	TblTemplate.InsertHParam(Table:= Table);          	
	Error													:= TblTemplate.Error;
	ErrorId													:= TblTemplate.ErrorId;
	ErrorText												:= TblTemplate.ErrorText;
	FilledRows												:= TblTemplate.FilledRows;
	
	SetHParam												:= NOT Error;
(*************************************************************************************)
END_METHOD

METHOD setPathDynamics : BOOL //Return value = TRUE if executed succesful
VAR_INPUT
	Acc,Dec,Jerk											:	LREAL;
END_VAR
	(* NCI SetPathDynamics schreiben						*)
	(*********************************************************)

(* Zielpos. in Tabelle schreiben ************************************************************)
	BlockCount 												:= BlockCount + 1;
	TblTemplate.PathDynamics.nDisplayIndex := LastBlockNo := SEL(BlockNo = 0, BlockNo, TableNumber * OffsetFactorTblNumber + BlockCount);

	TblTemplate.PathDynamics.fDec							:= Dec;
	TblTemplate.PathDynamics.fJerk							:= Jerk;
	TblTemplate.PathDynamics.fAcc							:= Acc;
                                                        	
	TblTemplate.InsertPathDynamics(Table:= Table);    	
	Error													:= TblTemplate.Error;
	ErrorId													:= TblTemplate.ErrorId;
	ErrorText												:= TblTemplate.ErrorText;
	FilledRows												:= TblTemplate.FilledRows;

	SetPathDynamics											:= NOT Error;
(***************************************************************************)
END_METHOD

METHOD setSParam : bool //Return value = TRUE if executed succesful
VAR_INPUT
	SParam													: UINT;
END_VAR
(* 														*)
(********************************************************)

(*************************************************************************************)
	BlockCount 												:= BlockCount + 1;
	TblTemplate.SParam.nDisplayIndex := LastBlockNo 		:= SEL(BlockNo = 0, BlockNo,  TableNumber * OffsetFactorTblNumber + BlockCount);
	TblTemplate.SParam.nSParam								:= SParam;
                                                        	
	TblTemplate.InsertSParam(Table:= Table);          	
	Error													:= TblTemplate.Error;
	ErrorId													:= TblTemplate.ErrorId;
	ErrorText												:= TblTemplate.ErrorText;
	FilledRows												:= TblTemplate.FilledRows;
	
	SetSParam												:= NOT Error;
(*************************************************************************************)
END_METHOD

METHOD setTangFollowingDesc : booL //Return value = TRUE if executed succesful
VAR_INPUT
    TangOn													: BOOL;
    TangAxis												: E_NciAxesInGroup;  
    PathAxis1												: E_NciAxesInGroup; 
    PathAxis2												: E_NciAxesInGroup; 
    Offset													: LREAL; 
    CriticalAngle1											: LREAL;
    TfBehavior												: E_TangentialFollowingBehavior; 
END_VAR
	(* NCI SetTangFollowingDesc schreiben						*)
	(*********************************************************)

(* Zielpos. in Tabelle schreiben ************************************************************)
	BlockCount 												:= BlockCount + 1;
	LastBlockNo 											:= SEL(BlockNo = 0, BlockNo, TableNumber * OffsetFactorTblNumber + BlockCount);

    TblTemplate.TangentialFollowingDesc.bTangOn				:= TangOn;
    TblTemplate.TangentialFollowingDesc.nTangAxis			:= TangAxis;
    TblTemplate.TangentialFollowingDesc.nPathAxis1			:= PathAxis1;
    TblTemplate.TangentialFollowingDesc.nPathAxis2			:= PathAxis2;
    TblTemplate.TangentialFollowingDesc.fOffset				:= Offset;
    TblTemplate.TangentialFollowingDesc.fCriticalAngle1		:= CriticalAngle1;
    TblTemplate.TangentialFollowingDesc.nTfBehavior			:= TfBehavior;
                       	
	TblTemplate.InsertTangFollowingDesc(Table:= Table);    	
	Error													:= TblTemplate.Error;
	ErrorId													:= TblTemplate.ErrorId;
	ErrorText												:= TblTemplate.ErrorText;
	FilledRows												:= TblTemplate.FilledRows;

	SetTangFollowingDesc									:= NOT Error;
(***************************************************************************)
END_METHOD

METHOD setTParam : bool //Return value = TRUE if executed succesful
VAR_INPUT
	TParam													: UINT;
END_VAR
(* 														*)
(********************************************************)

(*************************************************************************************)
	BlockCount 												:= BlockCount + 1;
	TblTemplate.TParam.nDisplayIndex := LastBlockNo 		:= SEL(BlockNo = 0, BlockNo,  TableNumber * OffsetFactorTblNumber + BlockCount);
	TblTemplate.TParam.nTParam								:= TParam;
                                                        	
	TblTemplate.InsertTParam(Table:= Table);          	
	Error													:= TblTemplate.Error;
	ErrorId													:= TblTemplate.ErrorId;
	ErrorText												:= TblTemplate.ErrorText;
	FilledRows												:= TblTemplate.FilledRows;
	
	SetTParam												:= NOT Error;
(**************************************************************************)
END_METHOD

METHOD setVertexSmoothing : BOOL //Return value = TRUE if executed succesful
VAR_INPUT
	Radius													: LREAL := 0.0;
	VertSmType												: UDINT := 5;
	VertSmSubType											: UDINT := 3;
END_VAR
(* writing NCI Vertex smoothing 								*)
(****************************************************************)

(* writing into table	*****************************************)
	BlockCount 												:= BlockCount + 1;
	TblTemplate.VertexSmoothing.nDisplayIndex := LastBlockNo := SEL(BlockNo = 0, BlockNo, TableNumber * OffsetFactorTblNumber + BlockCount);
	TblTemplate.VertexSmoothing.nType						:= VertSmType;
	TblTemplate.VertexSmoothing.nSubtype					:= VertSmSubtype; (* 	1: constant radius tolerance
																					2: distance between Abstand intersectoin point and peal point
																					3: adaptiv raidus tolerance
																					*)
	TblTemplate.VertexSmoothing.fRadius						:= Radius; (* mm *)

	TblTemplate.InsertVertexSmoothing(Table:= Table);
	Error													:= TblTemplate.Error;
	ErrorId													:= TblTemplate.ErrorId;
	ErrorText												:= TblTemplate.ErrorText;
	FilledRows												:= TblTemplate.FilledRows;
	SetVertexSmoothing										:= not Error;
(*************************************************************************************)
END_METHOD

END_FUNCTION_BLOCK

// POUs/Motion/TF5100-NCI/02_Options/PlcItp/NciCreateItpTableEntryTemplate
FUNCTION_BLOCK NciCreateItpTableEntryTemplate
VAR_INPUT
	EndOfTables												: ST_NciEndOfTables;
	GeoCirclePlane											: ST_NciGeoCirclePlane;
	GeoCircleCIP											: ST_NciGeoCircleCIP;
	GeoLine													: ST_NciGeoLine;
	GeoBezier3												: ST_NciGeoBezier3;
	GeoBezier5												: ST_NciGeoBezier5;	
	GeoStart												: ST_NciGeoStart;
	TangentialFollowingDesc									: ST_NciTangentialFollowingDesc;
	MFuncHsk												: ST_NciMFuncHsk;
	MFuncFast												: ST_NciMFuncFast;
	MFuncResetAllFast										: ST_NciMFuncResetAllFast;
	HParam													: ST_NciHParam;
	SParam													: ST_NciSParam;
	TParam													: ST_NciTParam;
	DynOverride												: ST_NciDynOvr;
	VertexSmoothing											: ST_NciVertexSmoothing;
	PathDynamics											: ST_NciPathDynamics;
	BaseFrame												: ST_NciBaseFrame;
	SetCoordinateSystem										: ST_NciSetCoordinateSystem;
	AxisDynamics											: ST_NciAxisDynamics;
	DwellTime												: ST_NciDwellTime;
END_VAR
VAR_OUTPUT
	FilledRows												: INT;
	Error													: BOOL;
{attribute 'displaymode':='hex'}
	ErrorId													: UDINT;
	ErrorText												: STRING(20);
END_VAR                 									
VAR                     									
	TblPrep													: FB_NciFeedTablePreparation;
END_VAR

(* NCI Table entry template				 	V2.0	*)
(****************************************************)

(******************************************************************************)
;
(******************************************************************************)

METHOD insertAxisDynamics : bool //Return value = TRUE if executed succesful
VAR_IN_OUT
	Table													: ST_NciFeedGroupTable;
END_VAR
	TblPrep(
		nEntryType			:= AxisDynamics.nEntryType,
		pEntry				:= ADR(AxisDynamics),
		stFeedGroupTable	:= Table,
		nFilledRows			=> FilledRows,
		bError				=> ,
		nErrorId			=> );

	IF TblPrep.bError 
	THEN
		Error												:= TRUE;
		ErrorText											:= CONCAT('AxisDynamics - JobNo. :',UDINT_TO_STRING(AxisDynamics.nDisplayIndex));
		ErrorId												:= TblPrep.nErrorId;
	ELSE
		insertAxisDynamics									:= TRUE;
	END_IF
END_METHOD

METHOD insertBaseFrame : bool //Return value = TRUE if executed succesful
VAR_IN_OUT
	Table													: ST_NciFeedGroupTable;
END_VAR
	TblPrep(
		nEntryType		:= BaseFrame.nEntryType,
		pEntry			:= ADR(BaseFrame),
		stFeedGroupTable:= Table,
		nFilledRows		=> FilledRows,
		bError			=> ,
		nErrorId		=> );

	IF TblPrep.bError 
	THEN
		Error												:= TRUE;
		ErrorText											:= CONCAT('BaseFrame - JobNo. :',UDINT_TO_STRING(BaseFrame.nDisplayIndex));
		ErrorId												:= TblPrep.nErrorId;
	ELSE
		insertBaseFrame										:= TRUE;
	END_IF
END_METHOD

METHOD insertDwellTime : booL //Return value = TRUE if executed succesful
VAR_IN_OUT
	Table													: ST_NciFeedGroupTable;
END_VAR
	TblPrep(
		nEntryType		:= DwellTime.nEntryType,
		pEntry			:= ADR(DwellTime),
		stFeedGroupTable:= Table,
		nFilledRows		=> FilledRows,
		bError			=> ,
		nErrorId		=> );

	IF TblPrep.bError 
	THEN
		Error												:= TRUE;
		ErrorText											:= CONCAT('DwellTime - JobNo. :',UDINT_TO_STRING(DwellTime.nDisplayIndex));
		ErrorId												:= TblPrep.nErrorId;
	ELSE
		insertDwellTime										:= TRUE;
	END_IF
END_METHOD

METHOD insertDynOverride : booL //Return value = TRUE if executed succesful
VAR_IN_OUT
	Table													: ST_NciFeedGroupTable;
END_VAR
	TblPrep(
		nEntryType			:= DynOverride.nEntryType,
		pEntry				:= ADR(DynOverride),
		stFeedGroupTable	:= Table,
		nFilledRows			=> FilledRows,
		bError				=> ,
		nErrorId			=> );

	IF TblPrep.bError THEN
		Error												:= TRUE;
		ErrorText											:= CONCAT('DynOverride - JobNo. :',UDINT_TO_STRING(DynOverride.nDisplayIndex));
		ErrorId												:= TblPrep.nErrorId;
	ELSE
		insertDynOverride									:= TRUE;
	END_IF
END_METHOD

METHOD insertEndOfTable : bool //Return value = TRUE if executed succesful
VAR_IN_OUT
	Table													: ST_NciFeedGroupTable;
END_VAR
	TblPrep(
		nEntryType			:= EndOfTables.nEntryType,
		pEntry				:= ADR(EndOfTables),
		stFeedGroupTable	:= Table,
		nFilledRows			=> FilledRows,
		bError				=> ,
		nErrorId			=> );

	IF TblPrep.bError THEN
		Error												:= TRUE;
		ErrorText											:= CONCAT('EndOfTables - FilledRows :',INT_TO_STRING(FilledRows));
		ErrorId												:= TblPrep.nErrorId;
	ELSE
		insertEndOfTable									:= TRUE;
	END_IF
END_METHOD

METHOD insertGeoBezier3 : booL //Return value = TRUE if executed succesful
VAR_IN_OUT
	Table													: ST_NciFeedGroupTable;
END_VAR
	TblPrep(
		nEntryType			:= GeoBezier3.nEntryType,
		pEntry				:= ADR(GeoBezier3),
		stFeedGroupTable	:= Table,
		nFilledRows			=> FilledRows,
		bError				=> ,
		nErrorId			=> );

	IF TblPrep.bError THEN
		Error												:= TRUE;
		ErrorText											:= CONCAT('GeoBezier3 - JobNo. :',UDINT_TO_STRING(GeoBezier3.nDisplayIndex));
		ErrorId												:= TblPrep.nErrorId;
	ELSE
		insertGeoBezier3									:= TRUE;
	END_IF
END_METHOD

METHOD insertGeoBezier5 : booL //Return value = TRUE if executed succesful
VAR_IN_OUT
	Table													: ST_NciFeedGroupTable;
END_VAR
	TblPrep(
		nEntryType			:= GeoBezier5.nEntryType,
		pEntry				:= ADR(GeoBezier5),
		stFeedGroupTable	:= Table,
		nFilledRows			=> FilledRows,
		bError				=> ,
		nErrorId			=> );

	IF TblPrep.bError THEN
		Error												:= TRUE;
		ErrorText											:= CONCAT('GeoBezier5 - JobNo. :',UDINT_TO_STRING(GeoBezier5.nDisplayIndex));
		ErrorId												:= TblPrep.nErrorId;
	ELSE
		insertGeoBezier5									:= TRUE;
	END_IF
END_METHOD

METHOD insertGeoCircleCIP : booL //Return value = TRUE if executed succesful
VAR_IN_OUT
	Table													: ST_NciFeedGroupTable;
END_VAR
	TblPrep(
		nEntryType			:= GeoCircleCIP.nEntryType,
		pEntry				:= ADR(GeoCircleCIP),
		stFeedGroupTable	:= Table,
		nFilledRows			=> FilledRows,
		bError				=> ,
		nErrorId			=> );

	IF TblPrep.bError 
	THEN
		Error												:= TRUE;
		ErrorText											:= CONCAT('GeoCircleCIP - JobNo. :',UDINT_TO_STRING(GeoCirclePlane.nDisplayIndex));
		ErrorId												:= TblPrep.nErrorId;
	ELSE
		insertGeoCircleCIP									:= TRUE;
	END_IF
END_METHOD

METHOD insertGeoCirclePlane : BOOL //Return value = TRUE if executed succesful
VAR_IN_OUT
	Table													: ST_NciFeedGroupTable;
END_VAR
	TblPrep(
		nEntryType			:= GeoCirclePlane.nEntryType,
		pEntry				:= ADR(GeoCirclePlane),
		stFeedGroupTable	:= Table,
		nFilledRows			=> FilledRows,
		bError				=> ,
		nErrorId			=> );

	IF TblPrep.bError 
	THEN
		Error												:= TRUE;
		ErrorText											:= CONCAT('GeoCirclePlane - JobNo. :',UDINT_TO_STRING(GeoCirclePlane.nDisplayIndex));
		ErrorId												:= TblPrep.nErrorId;
	ELSE
		insertGeoCirclePlane								:= TRUE;
	END_IF
END_METHOD

METHOD insertGeoLine : boOL //Return value = TRUE if executed succesful
VAR_IN_OUT
	Table													: ST_NciFeedGroupTable;
END_VAR
	TblPrep(
		nEntryType			:= GeoLine.nEntryType,
		pEntry				:= ADR(GeoLine),
		stFeedGroupTable	:= Table,
		nFilledRows			=> FilledRows,
		bError				=> ,
		nErrorId			=> );

	IF TblPrep.bError 
	THEN
		Error												:= TRUE;
		ErrorText											:= CONCAT('GeoLine - JobNo. :',UDINT_TO_STRING(GeoLine.nDisplayIndex));
		ErrorId												:= TblPrep.nErrorId;
	ELSE
		insertGeoLine										:= TRUE;
	END_IF
END_METHOD

METHOD insertGeoStart : booL //Return value = TRUE if executed succesful
VAR_IN_OUT
	Table													: ST_NciFeedGroupTable;
END_VAR
	TblPrep(
		nEntryType			:= GeoStart.nEntryType,
		pEntry				:= ADR(GeoStart),
		stFeedGroupTable	:= Table,
		nFilledRows			=> FilledRows,
		bError				=> ,
		nErrorId			=> );

	IF TblPrep.bError 
	THEN
		Error												:= TRUE;
		ErrorText											:= CONCAT('GeoStart - FilledRows. :',INT_TO_STRING(FilledRows));
		ErrorId												:= TblPrep.nErrorId;
	ELSE
		insertGeoStart										:= TRUE;
	END_IF
END_METHOD

METHOD insertHParam : booL //Return value = TRUE if executed succesful
VAR_IN_OUT
	Table													: ST_NciFeedGroupTable;
END_VAR
	TblPrep(
		nEntryType			:= HParam.nEntryType,
		pEntry				:= ADR(HParam),
		stFeedGroupTable	:= Table,
		nFilledRows			=> FilledRows,
		bError				=> ,
		nErrorId			=> );

	IF TblPrep.bError 
	THEN
		Error												:= TRUE;
		ErrorText											:= CONCAT('HParam - JobNo. :',UDINT_TO_STRING(HParam.nDisplayIndex));
		ErrorId												:= TblPrep.nErrorId;
	ELSE
		insertHParam										:= TRUE;
	END_IF
END_METHOD

METHOD insertMFuncFast : booL //Return value = TRUE if executed succesful
VAR_IN_OUT
	Table													: ST_NciFeedGroupTable;
END_VAR
	TblPrep(
		nEntryType			:= MFuncFast.nEntryType,
		pEntry				:= ADR(MFuncFast),
		stFeedGroupTable	:= Table,
		nFilledRows			=> FilledRows,
		bError				=> ,
		nErrorId			=> );

	IF TblPrep.bError 
	THEN
		Error												:= TRUE;
		ErrorText											:= CONCAT('MFuncFastList - JobNo. :',UDINT_TO_STRING(MFuncFast.nDisplayIndex));
		ErrorId												:= TblPrep.nErrorId;
	ELSE
		insertMFuncFast										:= TRUE;
	END_IF
END_METHOD

METHOD insertMFuncHsk : bool //Return value = TRUE if executed succesful
VAR_IN_OUT
	Table													: ST_NciFeedGroupTable;
END_VAR
	TblPrep(
		nEntryType			:= MFuncHsk.nEntryType,
		pEntry				:= ADR(MFuncHsk),
		stFeedGroupTable	:= Table,
		nFilledRows			=> FilledRows,
		bError				=> ,
		nErrorId			=> );

	IF TblPrep.bError 
	THEN
		Error												:= TRUE;
		ErrorText											:= CONCAT('MFuncHsk - JobNo. :',UDINT_TO_STRING(MFuncHsk.nDisplayIndex));
		ErrorId												:= TblPrep.nErrorId;
	ELSE
		insertMFuncHsk										:= TRUE;
	END_IF
END_METHOD

METHOD insertMFuncResetAllFast : bool //Return value = TRUE if executed succesful
VAR_IN_OUT
	Table													: ST_NciFeedGroupTable;
END_VAR
	TblPrep(
		nEntryType			:= MFuncResetAllFast.nEntryType,
		pEntry				:= ADR(MFuncResetAllFast),
		stFeedGroupTable	:= Table,
		nFilledRows			=> FilledRows,
		bError				=> ,
		nErrorId			=> );

	IF TblPrep.bError 
	THEN
		Error												:= TRUE;
		ErrorText											:= CONCAT('MFuncResetAllFast - JobNo. :',UDINT_TO_STRING(MFuncResetAllFast.nDisplayIndex));
		ErrorId												:= TblPrep.nErrorId;
	ELSE
		insertMFuncResetAllFast								:= TRUE;
	END_IF
END_METHOD

METHOD insertPathDynamics : BOOL //Return value = TRUE if executed succesful
VAR_IN_OUT
	Table													: ST_NciFeedGroupTable;
END_VAR
	TblPrep(
		nEntryType			:= PathDynamics.nEntryType,
		pEntry				:= ADR(PathDynamics),
		stFeedGroupTable	:= Table,
		nFilledRows			=> FilledRows,
		bError				=> ,
		nErrorId			=> );

	IF TblPrep.bError 
	THEN
		Error												:= TRUE;
		ErrorText											:= CONCAT('PathDynamics - JobNo. :',UDINT_TO_STRING(PathDynamics.nDisplayIndex));
		ErrorId												:= TblPrep.nErrorId;
	ELSE
		insertPathDynamics									:= TRUE;
	END_IF
END_METHOD

METHOD insertSetCoordinateSystem : bool //Return value = TRUE if executed succesful
VAR_IN_OUT
	Table													: ST_NciFeedGroupTable;
END_VAR
	TblPrep(
		nEntryType			:= SetCoordinateSystem.nEntryType,
		pEntry				:= ADR(SetCoordinateSystem),
		stFeedGroupTable	:= Table,
		nFilledRows			=> FilledRows,
		bError				=> ,
		nErrorId			=> );

	IF TblPrep.bError 
	THEN
		Error												:= TRUE;
		ErrorText											:= CONCAT('SetCoordinateSystem - JobNo. :',UDINT_TO_STRING(SetCoordinateSystem.nDisplayIndex));
		ErrorId												:= TblPrep.nErrorId;
	ELSE
		insertSetCoordinateSystem							:= TRUE;
	END_IF
END_METHOD

METHOD insertSParam : bool //Return value = TRUE if executed succesful
VAR_IN_OUT
	Table													: ST_NciFeedGroupTable;
END_VAR
	TblPrep(
		nEntryType			:= SParam.nEntryType,
		pEntry				:= ADR(SParam),
		stFeedGroupTable	:= Table,
		nFilledRows			=> FilledRows,
		bError				=> ,
		nErrorId			=> );

	IF TblPrep.bError 
	THEN
		Error												:= TRUE;
		ErrorText											:= CONCAT('SParam - JobNo. :',UDINT_TO_STRING(SParam.nDisplayIndex));
		ErrorId												:= TblPrep.nErrorId;
	ELSE
		insertSParam										:= TRUE;
	END_IF
END_METHOD

METHOD insertTangFollowingDesc : booL //Return value = TRUE if executed succesful
VAR_IN_OUT
	Table													: ST_NciFeedGroupTable;
END_VAR
	TblPrep(
		nEntryType			:= TangentialFollowingDesc.nEntryType,
		pEntry				:= ADR(TangentialFollowingDesc),
		stFeedGroupTable	:= Table,
		nFilledRows			=> FilledRows,
		bError				=> ,
		nErrorId			=> );

	IF TblPrep.bError 
	THEN
		Error												:= TRUE;
		ErrorText											:= CONCAT('TangentialFollowingDesc - JobNo. :','~');
		ErrorId												:= TblPrep.nErrorId;
	ELSE
		insertTangFollowingDesc								:= TRUE;
	END_IF
END_METHOD

METHOD insertTParam : bool //Return value = TRUE if executed succesful
VAR_IN_OUT
	Table													: ST_NciFeedGroupTable;
END_VAR
	TblPrep(
		nEntryType			:= TParam.nEntryType,
		pEntry				:= ADR(TParam),
		stFeedGroupTable	:= Table,
		nFilledRows			=> FilledRows,
		bError				=> ,
		nErrorId			=> );

	IF TblPrep.bError 
	THEN
		Error												:= TRUE;
		ErrorText											:= CONCAT('TParam - JobNo. :',UDINT_TO_STRING(TParam.nDisplayIndex));
		ErrorId												:= TblPrep.nErrorId;
	ELSE
		insertTParam										:= TRUE;
	END_IF
END_METHOD

METHOD insertVertexSmoothing : BOOL //Return value = TRUE if executed succesful
VAR_IN_OUT
	Table													: ST_NciFeedGroupTable;
END_VAR
	TblPrep(
		nEntryType			:= VertexSmoothing.nEntryType,
		pEntry				:= ADR(VertexSmoothing),
		stFeedGroupTable	:= Table,
		nFilledRows			=> FilledRows,
		bError				=> ,
		nErrorId			=> );

	IF TblPrep.bError 
	THEN
		Error												:= TRUE;
		ErrorText											:= CONCAT('VertexSmoothing - JobNo. :',UDINT_TO_STRING(VertexSmoothing.nDisplayIndex));
		ErrorId												:= TblPrep.nErrorId;
	ELSE
		insertVertexSmoothing								:= TRUE;
	END_IF
END_METHOD

METHOD reset : BOOL  //Return value = TRUE if execution finished
VAR_IN_OUT
	Table													: ST_NciFeedGroupTable;
END_VAR
TblPrep(
	nEntryType			:= ,
	pEntry				:= ,
	bResetTable			:= TRUE,
	bResetAll			:= TRUE,
	stFeedGroupTable	:= Table,
	nFilledRows			=> FilledRows,
	bError				=> ,
	nErrorId			=> );

TblPrep.bResetTable											:= FALSE;
TblPrep.bResetAll											:= FALSE;
Error														:= FALSE;
ErrorText													:= '';
ErrorId														:= 0;
Reset														:= TRUE;
END_METHOD

END_FUNCTION_BLOCK

// POUs/Motion/TF511x-KIN/03_DUTs/Trafo/UCS
{attribute 'hide'}
FUNCTION_BLOCK UCS
VAR_INPUT
	oid														:	UDINT := 0;		//Object identifier
	vTranslation 											:	VECTOR;
 	vRotation 												:	VECTOR;
	Valid													:	BOOL := FALSE;
END_VAR
VAR_OUTPUT
END_VAR
VAR
END_VAR

METHOD delete : BOOL
VAR_INPUT
END_VAR
MEMSET(ADR(vTranslation),0,SIZEOF(vTranslation));
MEMSET(ADR(VRotation),0,SIZEOF(VRotation));
oid 													:= 0;
delete	:= TRUE;
END_METHOD

END_FUNCTION_BLOCK

// POUs/Motion/TF5100-NCI/02_Options/RParameter/NCiReadWriteRParam
// To Start read or write, set inpult values and call action read/write. Busy and Done show the status of the operation
FUNCTION_BLOCK NCiReadWriteRParam EXTENDS FbBase
VAR_OUTPUT CONSTANT
	FNC_READ												:	INT := 0;
	FNC_WRITE												:	INT := 1;
END_VAR         											
VAR_INPUT       											
	Fnc														:	INT (FNC_READ..FNC_WRITE) := FNC_READ;
  	pAddr    												: 	DWORD; //Address of parameter destination variable
   	Index   												: 	DINT; //Index to parameter to read
   	Count   												: 	DINT; //
	rNCIRef													:	REFERENCE TO NCI_REF := 0;
END_VAR
VAR_OUTPUT
END_VAR
VAR
(* cache *******************************************************************)
	MemFnc													:	INT := -1;

(* trigger *****************************************************************)

(* function-block instances	************************************************)
	ItpReadRParamsEx										:	ItpReadRParamsEx := (tTimeout := DEFAULT_ADS_TIMEOUT);
	ItpWriteRParamsEx										:	ItpWriteRParamsEx := (tTimeout := DEFAULT_ADS_TIMEOUT);

END_VAR

	(* Read/Write Nci group R parameter													*)
	(************************************************************************************)

(* Execute ******************************************************************************)
	rtExecute(CLK := Execute);
	IF rtExecute.Q
		AND MemFnc < 0
	THEN
		MemFnc 												:= SEL(Fnc = FNC_WRITE, FNC_READ , FNC_WRITE) ;
		Busy												:= TRUE;
		Done												:= FALSE;
		Error												:= FALSE;
		ErrorID												:= 0;
	END_IF

(* Call Method ***************************************************************************)
	CASE MemFnc OF
	FNC_READ:
		Read(Execute );

	FNC_WRITE:
		Write(Execute );

	-1:
		IF NOT Execute
		THEN
			Busy											:= FALSE;
			Done											:= FALSE;
			Error											:= FALSE;
			ErrorID											:= 0;
		END_IF                              				
	ELSE                                    				
		Busy												:= FALSE;
		Done												:= FALSE;
		Error												:= Execute;
		ErrorID												:= E_AdsErr.DEVICE_INVALIDPARM;
	END_CASE

(*************************************************************************************************)

METHOD PUBLIC read : BOOL //Return value = TRUE if busy
//required parameter
//pAddr
//Index
//Count
//rNCIRef
VAR_INPUT 
	Execute													:	BOOL;
END_VAR
	MemFnc 													:= FNC_READ;
	This^.Execute											:= Execute;
IF NOT __ISVALIDREF(rNCIRef) OR pAddr = 0 
THEN
	Busy													:= NOT Error;
	ErrorId													:= E_adsErr.DEVICE_INVALIDPARM;
	Error													:= TRUE;
	Done													:= FALSE;
	MemFnc													:= SEL(Execute , -1 ,MemFnc); 
	RETURN;
END_IF
	
	IF Execute
	THEN
		Error												:=	FALSE;
		ErrorId												:= 0;
		ItpReadRParamsEx.bExecute 							:= TRUE;
	ELSIF NOT ItpReadRParamsEx.bBusy    					
	THEN                                					
		Error												:=	FALSE;
		ErrorId												:= 0;
		ItpReadRParamsEx.bExecute 							:= FALSE;

	END_IF

	ItpReadRParamsEx(
		bExecute	:= ,
		pAddr		:= pAddr,
		nIndex		:= Index,
		nCount		:= Count,
		tTimeOut	:= ,
		sNciToPlc	:= rNCIRef.NciToPlc,
		bBusy		=> Busy,
		bErr		=> ,
		nErrId		=> );

	Done													:= NOT ItpReadRParamsEx.bBusy
																AND NOT ItpReadRParamsEx.bErr
																AND ItpReadRParamsEx.bExecute;
                                                        	
	IF NOT Busy                                         	
	THEN                                                	
		IF ItpReadRParamsEx.bExecute                    	
		THEN                                            	
			Error											:=	ItpReadRParamsEx.bErr;
			ErrorId											:= ItpReadRParamsEx.nErrId;
		END_IF                          					
		IF NOT Execute                  					
		THEN                            	            	
			MemFnc											:= -1;
			ItpReadRParamsEx(bExecute := FALSE , sNciToPlc:= rNCIRef.NciToPlc);
		END_IF
	END_IF
	
	read													:= Busy;
END_METHOD

METHOD PUBLIC write : BOOL //Return value = TRUE if busy
//required parameter
//pAddr
//Index
//Count
//rNCIRef
VAR_INPUT
	Execute													:	BOOL;
END_VAR
	MemFnc 													:= FNC_WRITE;
	THIS^.Execute											:= Execute;

IF NOT __ISVALIDREF(rNCIRef) OR pAddr = 0 
THEN
	Busy													:= NOT Error;
	ErrorId													:= E_adsErr.DEVICE_INVALIDPARM;
	Error													:= TRUE;
	Done													:= FALSE;
	MemFnc													:= SEL(Execute , -1 ,MemFnc); 
	RETURN;
END_IF

	IF Execute
	THEN
		Error												:=	FALSE;
		ErrorId												:= 0;
		ItpWriteRParamsEx.bExecute 							:= TRUE;
	ELSIF NOT ItpWriteRParamsEx.bBusy   					
	THEN                                					
		Error												:=	FALSE;
		ErrorId												:= 0;
		ItpWriteRParamsEx.bExecute 							:= FALSE;

	END_IF

	ItpWriteRParamsEx(
		bExecute	:= ,
		pAddr		:= pAddr,
		nIndex		:= Index,
		nCount		:= Count,
		tTimeOut	:= ,
		sNciToPlc	:= rNCIRef.NciToPlc,
		bBusy		=> Busy,
		bErr		=> ,
		nErrId		=> );

	Done													:= NOT ItpWriteRParamsEx.bBusy
																AND NOT ItpWriteRParamsEx.bErr
																AND ItpWriteRParamsEx.bExecute;
                                        					
	IF NOT Busy
	THEN
		IF ItpWriteRParamsEx.bExecute
		THEN
			Error											:=	ItpWriteRParamsEx.bErr;
			ErrorId											:= ItpWriteRParamsEx.nErrId;
		END_IF                          					
		IF NOT Execute                  					
		THEN                            	
			MemFnc											:= -1;
			ItpWriteRParamsEx(bExecute := FALSE, sNciToPlc:= rNCIRef.NciToPlc);
		END_IF
	END_IF
	
	write													:= Busy;
END_METHOD

END_FUNCTION_BLOCK

// POUs/Motion/TF5100-NCI/NciChannel
{attribute 'no_check'}
FUNCTION_BLOCK NciChannel EXTENDS NCI_REF
VAR_INPUT
	Admin													:	NciAdmin;
	grp														:	NciGrp;
	Itp														:	NciItp;
	motion													:	NciMotion;
                        								   
	MFnc													: 	NciMFnc;
	RPara													:	NciReadWriteRParam;
                        								      
	Event													:	NciEventHandling;
                        	
END_VAR                 	
VAR_OUTPUT              	
	ErrHdl													:	ERROR_HDL;
END_VAR
VAR
END_VAR

	(* NCI Control											*)
	(********************************************************)

(********************************************************************************)
(* error event ctrl																*)
(********************************************************************************)
	Event(
		Enable			:= ,
		ConfirmTrig		:= NOT Errhdl.flag AND Event.Status.31 OR Admin.ResetAdmin,
		Name			:= ErrHdl.fnc,
		SourceId		:= (* Default *) ,
		rNci			:= THIS^,
		ErrorId			:= TO_UDINT(ErrHdl.Id),
		Status			=> );
		
	(* Reset FB errors by reset flag *)
	(* currently not in use, call _Resetting via state machine to reset Fb errors by setting Execute to FALSE 
	IF Admin.Reset
	THEN
		grp.Execute											:= grp.Execute AND NOT grp.Error;
		itp.Execute											:= itp.Execute AND NOT itp.Error;
		Motion.Execute										:= Motion.Execute AND NOT Motion.Error;
		RPara.Execute										:= RPara.Execute AND NOT RPara.Error;
	END_IF
	*)
	
(********************************************************************************)
(* work admin ctrl																*)
(********************************************************************************)
	admin(
		ResetAdmin					:= ,
		Enable					:= ,
		EStop					:= ,
		SingleBlockMode			:= , 
		InSingleBlockTrigNext	:= , 
		GrpCnfg					:= ,
		Override				:= ,
		SpindleOvr				:= ,	
		rNCIRef					:= THIS^,
		InGroup					=> ,
		Busy					=> ,
		Done					=> ,
		Error					=> ,
		ErrorID					=> ,
		ErrorText				=> );

(********************************************************************************)
(* work group ctrl																*)
(********************************************************************************)
	grp(
		Execute				:= ,
		Fnc					:= ,
		XAxisId				:= ,
		YAxisId				:= ,
		ZAxisId				:= ,
		Q1AxisId			:= ,
		Q2AxisId			:= ,
		Q3AxisId			:= ,
		Q4AxisId			:= ,
		Q5AxisId			:= ,
		AxisIndex			:= ,
		rNCIRef				:= THIS^, 
		Busy				=> ,
		Done				=> ,
		Error				=> ,
		ErrorID				=> ,
		ErrorText			=> );

(********************************************************************************)
(* work interpolation ctrl														*)
(********************************************************************************)
	Itp(
		Execute				:= ,
		Fnc					:= ,
		Prg					:= ,
		rTable				:= ,
		rNCIRef				:= THIS^,
		StartPrgAfterLoading:= , 
		LogFeederEntries	:= ,
		Busy				=> ,
		Done				=> ,
		Error				=> ,
		ErrorID				=> ,
		ErrorText			=> );


(********************************************************************************)
(* work motion ctrl																*)
(********************************************************************************)
	motion(
		Execute						:= ,
		Fnc							:= ,
		rNCIRef						:= THIS^,
		FNC_ESTOP					=> ,
		FNC_STEP_ON					=> ,
		FNC_ENABLE_FEEDER_BACKUP	=> ,
		FNC_DISABLE_FEEDER_BACKUP	=> ,
		FNC_RETRACE_FWD				=> ,
		FNC_RETRACE_BWD				=> ,
		Busy						=> ,
		Done						=> ,
		Error						=> ,
		ErrorId						=> ,
		ErrorText					=> );

(********************************************************************************)
(* work R rarameter ctrl														*)
(********************************************************************************)
	RPara(
		Execute						:= ,
		Fnc							:= ,
		pAddr						:= ,
		Index						:= ,
		Count						:= ,
		rNCIRef						:= THIS^,
		Done						=> ,
		Busy						=> ,
		Error						=> ,
		ErrorId						=> );

(********************************************************************************)
(* work M function  ctrl														*)
(********************************************************************************)
	MFnc(
		ConfirmHsk					:= ,
		FastMFuncReset				:= ,
		FastMFuncNo					:= ,
		rNCIRef						:= THIS^);

(********************************************************************************)
(* collect errors																*)
(********************************************************************************)
	IF Admin.Error
	THEN
		ErrHdl.flag											:= Admin.Error;
		ErrHdl.id											:= UDINT_TO_DINT(Admin.ErrorID);
		ErrHdl.fnc											:= 'NciAdmin';
		ErrHdl.text											:= Admin.ErrorText;
                        									
	ELSIF grp.Error     									
	THEN                									
		ErrHdl.flag											:= grp.Error;
		ErrHdl.id											:= UDINT_TO_DINT(grp.ErrorID);
		ErrHdl.fnc											:= 'NciGrp';
		ErrHdl.text											:= grp.ErrorText;
                        									
	ELSIF itp.Error     									
	THEN                									
		ErrHdl.flag											:= Itp.Error;
		ErrHdl.id											:= UDINT_TO_DINT(Itp.ErrorID);
		ErrHdl.fnc											:= 'NciItp';
		ErrHdl.text											:= Itp.ErrorText;
                        									
	ELSIF motion.Error  									
	THEN                									
		ErrHdl.flag											:= motion.Error;
		ErrHdl.id											:= UDINT_TO_DINT(motion.ErrorID);
		ErrHdl.fnc											:= 'NciMotion';
		ErrHdl.text											:= motion.ErrorText;
		
	ELSIF RPara.Error  									
	THEN                									
		ErrHdl.flag											:= RPara.Error;
		ErrHdl.id											:= UDINT_TO_DINT(RPara.ErrorID);
		ErrHdl.fnc											:= 'RPara';
		ErrHdl.text											:= CONCAT('Error RPara id: ',  UDINT_TO_STRING(RPara.Errorid));
	ELSE
		ErrHdl.Reset();
	END_IF
(******************************************************************************)

METHOD PUBLIC noAction : BOOL
VAR_INPUT
END_VAR
grp.Execute													:= FALSE;
itp.Execute													:= FALSE;
Motion.Execute												:= FALSE;
RPara.Execute												:= FALSE;

NoAction 													:= NOT Grp.Busy and not Itp.Busy and not Motion.Busy and not RPara.Busy;
END_METHOD

METHOD reset : Bool
VAR_INPUT
END_VAR
NoAction();
reset 			:= ErrHdl.flag OR Admin.reset(FALSE);
Event.confirm();
END_METHOD

END_FUNCTION_BLOCK

// POUs/Motion/TF511x-KIN/01_Main/KIN_REF
//Kinematic group ref - call ReadStatus cyclic
FUNCTION_BLOCK KIN_REF
VAR_INPUT
	PlcToNci										AT %Q*	:	PLCTONC_NCICHANNEL_REF;
END_VAR                     						
VAR_OUTPUT                  						
	NciToPlc										AT %I*	:	NCTOPLC_NCICHANNEL_REF;
                            						
	ChnOperationState										:	E_KINSTATUS := 0;
	CartesianModeON											:	BOOL := FALSE;
	                                					
(* ChnState ***************************)
	IsKinematicChn											:	BOOL := FALSE;
	                                					
	AxList													: ST_KinAxes;
END_VAR
VAR
END_VAR

;

METHOD PUBLIC readStatus : booL;
VAR_INPUT
END_VAR
(* Kin Channel State *********************************************************)
	F_KinGetAcsMcsAxisIds(AxList,NciToPlc);
	
	ChnOperationState 										:= TO_INT(F_KinGetChnOperationState(NciToPlc));

	CartesianModeON											:= NciToPlc.AcsAxisIDs[0] <> 0 AND NciToPlc.AcsAxisIDs[1] <> 0;
	
	IsKinematicChn											:= NciToPlc.ChnState.1;

	readStatus												:= TRUE;
(*****************************************************************************)
END_METHOD

END_FUNCTION_BLOCK

// POUs/Motion/TF511x-KIN/01_Main/KinAdmin
//Kinematic group administration - Enable/Disable/Reset group
//based on TF511x - Tc2_NcKinematicTransformation
//ACS - Axis coordinate system => Robot motors M1-Mx 
//MCS - Machine coordinate system >= Cartesian Axis X,Y,Z,Rx,Ry,Rz (A,B,C) 
FUNCTION_BLOCK KinAdmin
VAR_INPUT
	ResetTrig												:	BOOL := FALSE;
	Enable													:	BOOL := FALSE; (* TRUE = Build Group , FALSE = Reconfig Group *)
	Override												:	LREAL	:= 0.0;
	ItpChannelId 											: 	UDINT := 0; (* Bei 0 wirtd der ITP Kanal nicht resetet *)
	AxesList												: 	ST_KinAxes;
	rKINRef													:	REFERENCE TO KIN_REF := 0;
END_VAR
VAR_IN_OUT
END_VAR
VAR_OUTPUT
	Busy													:	BOOL;
	Done													:	BOOL;
	Error													:	BOOL;
{attribute 'displaymode':='hex'}
	ErrorId													:	UDINT;
	ErrorText												:	STRING(40);
END_VAR
VAR
(* cache **************************************************************************)
	MemDone													:	BOOL;
	MemFnc													:	INT := 1;
	                        								
(* MC-functonblock instances *******************************************************)
	ResetKinGroup											: 	FB_KinResetGroup ;
	ConfigKinGroup											:	FB_KinConfigGroup  ;

(* Dummy Speicher **********************************************************)
	OK 														: BOOL;
END_VAR

	(* Kinematic group administration										*)
	(************************************************************************)

(* aborting function-block call if pointer is not valid ****************************************)
IF NOT __ISVALIDREF(rKINRef) 
THEN
	Busy													:= NOT Error;
	ErrorId													:= E_AdsErr.DEVICE_INVALIDPARM;
	Error													:= TRUE;
	Done													:= FALSE;
	ErrorText												:= 'Reference to rKINRef invalid (0)';
	RETURN;
END_IF

(* reading axis-status from NCtoPLC-channel ***************************************************)
	rKINRef.readStatus();

(* accepting setvalue-barrier e.g. for hardware limit switch **********************************)
	rKINRef.PlcToNci.ChnAxesOvr 							:= LREAL_TO_DWORD(LIMIT(0.0,Override,100.0) * 10000.0 );

(* ctrl programm ******************************************************************************)
	ConfigKinGroup.bExecute									:=	NOT ConfigKinGroup.bBusy
																AND(
																Enable
																AND NOT ConfigKinGroup.bCartesianMode
																OR
																NOT Enable
																AND ConfigKinGroup.bCartesianMode);

	IF ConfigKinGroup.bExecute
	THEN
		ConfigKinGroup.bCartesianMode						:= Enable;
	END_IF

	ConfigKinGroup(
		bExecute		:= ,
		bCartesianMode	:= ,
		stAxesList		:= AxesList,
		stKinRefIn		:= rKinRef.NciToPlc,
		bBusy			=> ,
		bDone			=> ,
		bError			=> ,
		nErrorId		=> );

(* Reset Grp ****************************************************************)
	IF Memfnc < 0
	THEN
		IF ResetTrig
		THEN
			reset(Execute:= TRUE);
			MemFnc											:= 1;
		END_IF
	ELSIF NOT reset(Execute:= ResetTrig)
	THEN
		MemFnc												:= -1;
	END_IF

(******************************************************************************)
(* Ctrl Status 																					*)
(******************************************************************************)
	Busy						:= ResetKinGroup.bBusy OR ConfigKinGroup.bBusy;
	
	IF Busy
	THEN
		Error												:= FALSE;
		ErrorId												:= 0;
		ErrorText											:= '';
	ELSIF ConfigKinGroup.bError
	THEN
		Error												:= TRUE;
		ErrorId												:= ConfigKinGroup.nErrorID;
		ErrorText											:= CONCAT('ConfigKinGroup ErrorId: ', UDINT_TO_STRING(Errorid));
	ELSIF ResetKinGroup.bExecute
		AND ResetKinGroup.bError
	THEN
		Error												:= TRUE;
		ErrorId												:= ResetKinGroup.nErrorID;
		ErrorText											:= CONCAT('ResetKinGroup ErrorId: ', UDINT_TO_STRING(Errorid));
	ELSIF rKINRef.NciToPlc.ErrorCode <> 0
	THEN
		Error												:= TRUE;
		ErrorId												:= rKINRef.NciToPlc.ErrorCode;
		ErrorText											:= CONCAT('KIN Grp ErrorId: ', UDINT_TO_STRING(Errorid));
	ELSE
		Error												:= FALSE;
		ErrorId												:= 0;
		ErrorText											:= '';
	END_IF

	IF ResetKinGroup.bDone
		OR ConfigKinGroup.bDone
	THEN
		MemDone												:= TRUE;
	END_IF

	Done													:= NOT Busy AND MemDone;

	IF done
	THEN
		MemDone												:= FALSE;
	END_IF

(**************************************************************************************************)

METHOD PUBLIC reset : BOOL //Return value = TRUE if busy
//required parameter
//rKinRef
//ItpChannelId
//AxesList
VAR_INPUT
	Execute													:	BOOL;
END_VAR
IF NOT __ISVALIDREF(rKINRef) THEN
	Busy													:= NOT Error;
	ErrorId													:=E_AdsErr.DEVICE_INVALIDPARM;
	Error													:= TRUE;
	Done													:= FALSE;
	ErrorText												:= 'Reference to rKINRef  invalid (0)';
	RETURN;
END_IF

	IF Execute
	THEN
		Error												:=	FALSE;
		ErrorId												:= 0;
		ResetKinGroup.bExecute 								:= rKinRef.NciToPlc.ErrorCode <> 0;
	ELSIF NOT ResetKinGroup.bBusy
	THEN
		Error												:=	FALSE;
		ErrorId												:= 0;
		ResetKinGroup.bExecute 								:= FALSE;

	END_IF

	ResetKinGroup(
		bExecute		:= ,
		nItpChannelId	:= ItpChannelId,
		stKinRefIn		:= rKinRef.NciToPlc,
		stAxesList		:= AxesList,
		bBusy			=> Busy,
		bDone			=> ,
		bError			=> ,
		nErrorId		=> );

	Done													:= NOT ResetKinGroup.bBusy
																AND NOT ResetKinGroup.bError
																AND ResetKinGroup.bExecute;

	IF NOT Busy
	THEN
		IF ResetKinGroup.bExecute
		THEN
			Error											:=	ResetKinGroup.bError;
			ErrorId											:= ResetKinGroup.nErrorId;
			ErrorText										:= SEL(Error , '' ,  CONCAT('Error ResetKinGroup id: ',  UDINT_TO_STRING(Errorid)));
		END_IF
		IF NOT Execute
		THEN
			MemFnc											:= -1 ;
			ResetKinGroup(	bExecute := FALSE, 
							stKinRefIn := rKinRef.NciToPlc, 
							stAxesList := AxesList);
		END_IF
	END_IF
	
	reset													:= Busy;
END_METHOD

END_FUNCTION_BLOCK

// POUs/Motion/TF511x-KIN/02_Options/KinLockUnlockTrafoParam
//Lock or Unlock kinematic group parameter
FUNCTION_BLOCK KinLockUnlockTrafoParam
VAR_INPUT
	Execute													:	BOOL	:= FALSE;
	Lock													:	BOOL 	:= TRUE;
   	oidTrafo												:	UDINT;
END_VAR                     								
VAR_OUTPUT                  								
	Busy													:	BOOL	:= FALSE;
	Done													:	BOOL	:= FALSE;
	Error													:	BOOL	:= FALSE;
	ErrorId													:	UDINT	:= 0;
END_VAR                     								
VAR                         	
	State													:	UDINT	:= 0;
	ADSWRITE												:	ADSWRITE;
END_VAR

CASE State OF
0:
	Done													:= FALSE;
	Error													:= FALSE;
	ErrorId													:= 0;
	Busy 													:= FALSE;
	
	IF Execute THEN
		AdsWrite(WRITE := FALSE);
		AdsWrite(
			NETID		:='',
			PORT		:= 10,
			IDXGRP		:=oidTrafo,
			IDXOFFS		:=SEL(Lock, 16#05030210, 16#0503020F),
			LEN			:= 0,
			SRCADDR		:=0 ,
			WRITE		:= TRUE,
			TMOUT		:= DEFAULT_ADS_TIMEOUT,
			BUSY		=> ,
			ERR			=> ,
			ERRID		=> );

		Busy												:= TRUE;
		State												:= 10;
	END_IF
10:
	AdsWrite(
		TMOUT	:= DEFAULT_ADS_TIMEOUT,
		BUSY	=>,
		ERR		=>Error,
		ERRID	=>ErrorId);
		
	IF NOT AdsWrite.BUSY 
	THEN
		IF NOT AdsWrite.ERR 
		THEN
			Done											:= TRUE;
		END_IF
		IF NOT Execute THEN
			State											:= 0;
		ELSE
			State											:= 20;
		END_IF
		AdsWrite(WRITE:=FALSE);
	END_IF
20:
	Busy													:= FALSE;
	IF NOT Execute THEN
		State												:= 0;
	END_IF

END_CASE

END_FUNCTION_BLOCK

// POUs/Motion/TF511x-KIN/02_Options/KinWriteToolTrafoParam
{attribute 'hide'}
(*==============================================================================*)
(* Name:			KIN_WriteToolTrafoParam							  	 		*)
(* Desc:			THIS IS NOT A RELEASED IMPLEMENTATION AND    				*)
(*  	           	SUBJECT TO CHANGE                            				*)
(*     			 															    *)
(* Author:	 	DS																*)
(* Date:							     										*)
(*==============================================================================*)
FUNCTION_BLOCK KinWriteToolTrafoParam
VAR_INPUT
	Execute													:	BOOL	:= FALSE;
   	oidTrafo												:	UDINT;
	ToolX													:	LREAL := 0.0;
	ToolY													:	LREAL := 0.0;
	ToolZ													:	LREAL := 0.0;
END_VAR                     								
VAR_OUTPUT                  								
	Busy													:	BOOL	:= FALSE;
	Done													:	BOOL	:= FALSE;
	Error													:	BOOL	:= FALSE;
	ErrorId													:	UDINT	:= 0;
END_VAR
VAR
	State													:	UDINT	:= 0;
	ADSWRITE												:ADSWRITE;
END_VAR

CASE State OF
0:
	Done													:= FALSE;
	Busy 													:= FALSE;
	Error													:= FALSE;
	ErrorId													:= 0;
	IF Execute 
	THEN
		AdsWrite(WRITE := FALSE);
		AdsWrite(
			NETID	:='',
			PORT	:= 10,
			IDXGRP	:=oidTrafo,
			IDXOFFS	:=SEL(FALSE (* Lock *), 16#05030210, 16#0503020F),
			LEN		:= 0,
			SRCADDR	:=0 ,
			WRITE	:= TRUE,
			TMOUT	:= DEFAULT_ADS_TIMEOUT,
			BUSY	=> ,
			ERR		=> ,
			ERRID	=> );

		Busy												:= TRUE;
		State												:= 1;
	END_IF

1:
	AdsWrite(
		TMOUT	:= DEFAULT_ADS_TIMEOUT,
		BUSY	=>,
		ERR		=>Error,
		ERRID	=>ErrorId);
		
	IF NOT AdsWrite.BUSY 
	THEN
		AdsWrite(WRITE:=FALSE);
			
		IF NOT AdsWrite.ERR 
		THEN
			AdsWrite( (* Write Tool X *)
				NETID	:= '',
				PORT	:= 10,
				IDXGRP	:= oidTrafo, 				(*OID 	Tool trafo*)
				IDXOFFS	:= 16#05010020, 			(*PTCID	Tool Trafo Parameter*)
				LEN		:= SIZEOF(ToolX),
				SRCADDR	:= ADR(ToolX),
				TMOUT	:= DEFAULT_ADS_TIMEOUT,
				WRITE 	:= TRUE,
				BUSY	=> ,
				ERR		=> ,
				ERRID	=> );
	

			State											:= 10;
		ELSE
			IF NOT Execute
			THEN
				State										:= 0;
			ELSE
				State										:= 99;
			END_IF
		END_IF
	END_IF

10:
	AdsWrite(
		TMOUT	:= DEFAULT_ADS_TIMEOUT,
		BUSY	=>,
		ERR		=>Error,
		ERRID	=>ErrorId);
		
	IF NOT AdsWrite.BUSY 
	THEN
		AdsWrite(WRITE:=FALSE);
		
		IF NOT AdsWrite.ERR 
		THEN
			AdsWrite( 								(* Write Tool Y *)
				NETID	:= '',
				PORT	:= 10,
				IDXGRP	:= oidTrafo, 				(*OID 	Tool trafo*)
				IDXOFFS	:= 16#05010021, 			(*PTCID	Tool Trafo Parameter*)
				LEN		:= SIZEOF(ToolY),
				SRCADDR	:= ADR(ToolY),
				TMOUT	:= DEFAULT_ADS_TIMEOUT,
				WRITE	:= TRUE,
				BUSY	=> ,
				ERR		=> ,
				ERRID	=> );

			State											:= 20;
		ELSE
			State											:= 90;
		END_IF
	END_IF

20:
	AdsWrite(
		TMOUT	:= DEFAULT_ADS_TIMEOUT,
		BUSY	=>,
		ERR		=>Error,
		ERRID	=>ErrorId);

	IF NOT AdsWrite.BUSY 
	THEN
		AdsWrite(WRITE:=FALSE);
		
	IF NOT AdsWrite.ERR 
	THEN
			AdsWrite( 								(* Write Tool Z *)
				NETID	:= '',
				PORT	:= 10,
				IDXGRP	:= oidTrafo, 				(*OID 	Tool trafo*)
				IDXOFFS	:= 16#05010022, 			(*PTCID	Tool Trafo Parameter*)
				LEN		:= SIZEOF(ToolZ),
				SRCADDR	:= ADR(ToolZ),
				TMOUT	:= DEFAULT_ADS_TIMEOUT,
				WRITE 	:= TRUE,
				BUSY	=> ,
				ERR		=> ,
				ERRID	=> );

			State											:= 60;
		ELSE            									
			State											:= 90;
		END_IF
	END_IF

60:
	AdsWrite(
		TMOUT	:= DEFAULT_ADS_TIMEOUT,
		BUSY	=>,
		ERR		=>Error,
		ERRID	=>ErrorId);

	IF NOT AdsWrite.BUSY 
	THEN
		State												:= 90;
		AdsWrite(WRITE:=FALSE);
	END_IF


90: (* Start Lock-Param *)
	AdsWrite(
		NETID	:='',
		PORT	:= 10,
		IDXGRP	:=oidTrafo,
		IDXOFFS	:=SEL(TRUE (* Lock *), 16#05030210, 16#0503020F),
		LEN		:= 0,
		SRCADDR	:=0 ,
		WRITE	:= TRUE,
		TMOUT	:= DEFAULT_ADS_TIMEOUT,
		BUSY	=> ,
		ERR		=> ,
		ERRID	=> );

	State													:= 91;

91:
	AdsWrite(
		TMOUT	:= DEFAULT_ADS_TIMEOUT,
		BUSY	=>,
		ERR		=>,
		ERRID	=>);

	IF NOT AdsWrite.BUSY 
	THEN
		Busy 												:= FALSE;
		IF NOT AdsWrite.ERR 
		THEN
			Done											:= NOT Error;
		ELSIF NOT Error
		THEN
			Error 											:= AdsWrite.ERR;
			ErrorId 										:= AdsWrite.ERRID;
		END_IF
		IF NOT Execute 
		THEN
			State											:= 0;
		ELSE        										
			State											:= 99;
		END_IF
		AdsWrite(WRITE:=FALSE);
	END_IF

99:
	Busy													:= FALSE;
	IF NOT Execute THEN
		State												:= 0;
	END_IF

END_CASE

END_FUNCTION_BLOCK

// POUs/Motion/TF511x-KIN/02_Options/KinWriteUCSTrafoParam
{attribute 'hide'}
(*==============================================================================*)
(* Name:			KIN_WriteUCSTrafoParam							  	 		*)
(* Desc:			THIS IS NOT A RELEASED IMPLEMENTATION AND    				*)
(*  	           	SUBJECT TO CHANGE                            				*)
(*     			 															    *)
(* Author:	 	DS																*)
(* Date:							     										*)
(*==============================================================================*)
FUNCTION_BLOCK KinWriteUCSTrafoParam
VAR_INPUT
	Execute													:	BOOL	:= FALSE;
   oidTrafo													:	UDINT;
	vTranslation 											:	VECTOR;
 	vRotation 												:	VECTOR;
END_VAR
VAR_OUTPUT
	Busy													:	BOOL	:= FALSE;
	Done													:	BOOL	:= FALSE;
	Error													:	BOOL	:= FALSE;
	ErrorId													:	UDINT	:= 0;
END_VAR
VAR
	State													:	UDINT	:= 0;
	ADSWRITE												:ADSWRITE;
END_VAR

CASE State OF
0:
	Done													:= FALSE;
	Busy													:= FALSE;
	Error													:= FALSE;
	ErrorId													:= 0;
	IF Execute 
	THEN
		AdsWrite(WRITE := FALSE);
		AdsWrite(
			NETID	:='',
			PORT	:= 10,
			IDXGRP	:=oidTrafo,
			IDXOFFS	:=SEL(FALSE (* Lock *), 16#05030210, 16#0503020F),
			LEN		:= 0,
			SRCADDR	:=0 ,
			WRITE	:= TRUE,
			TMOUT	:= DEFAULT_ADS_TIMEOUT,
			BUSY	=> ,
			ERR		=> ,
			ERRID	=> );

		Busy												:= TRUE;
		State												:= 1;
	END_IF

1: (* Start Translation X *)
	AdsWrite(
		TMOUT	:= DEFAULT_ADS_TIMEOUT,
		BUSY	=>,
		ERR		=>Error,
		ERRID	=>ErrorId);
		
	IF NOT AdsWrite.BUSY 
	THEN
		AdsWrite(WRITE:=FALSE);
		IF NOT AdsWrite.ERR 
		THEN
			AdsWrite(
				NETID	:= '',
				PORT	:= 10,
				IDXGRP	:= oidTrafo,
				IDXOFFS	:= 16#05010020,
				LEN		:= SIZEOF(vTranslation.m[1]),
				SRCADDR	:= ADR(vTranslation.m[1]),
				TMOUT	:= DEFAULT_ADS_TIMEOUT,
				WRITE 	:= TRUE,
				BUSY	=> ,
				ERR		=> ,
				ERRID	=> );

			State											:= 10;
		ELSE (* Error unlock Param *)
			IF NOT Execute 
			THEN
				State										:= 0;
			ELSE
				State										:= 99;
			END_IF
		END_IF
	END_IF

10: (* Translation Y *)
	AdsWrite(
		TMOUT	:= DEFAULT_ADS_TIMEOUT,
		BUSY	=>,
		ERR		=>Error,
		ERRID	=>ErrorId);
		
	IF NOT AdsWrite.BUSY 
	THEN
		AdsWrite(WRITE:=FALSE);
		
		IF NOT AdsWrite.ERR 
		THEN
			AdsWrite(
				NETID	:= '',
				PORT	:= 10,
				IDXGRP	:= oidTrafo,
				IDXOFFS	:= 16#05010021,
				LEN		:= SIZEOF(vTranslation.m[2]),
				SRCADDR	:= ADR(vTranslation.m[2]),
				TMOUT	:= DEFAULT_ADS_TIMEOUT,
				WRITE 	:= TRUE,
				BUSY	=> ,
				ERR		=> ,
				ERRID	=> );

			State											:= 20;
		ELSE            									
			State											:= 90;
		END_IF

	END_IF

20: (* Translation Z *)
	AdsWrite(
		TMOUT	:= DEFAULT_ADS_TIMEOUT,
		BUSY	=>,
		ERR		=>Error,
		ERRID	=>ErrorId);

	IF NOT AdsWrite.BUSY 
	THEN
		AdsWrite(WRITE:=FALSE);
		IF NOT AdsWrite.ERR 
		THEN
			AdsWrite(
				NETID	:= '',
				PORT	:= 10,
				IDXGRP	:= oidTrafo,
				IDXOFFS	:= 16#05010022,
				LEN		:= SIZEOF(vTranslation.m[3]),
				SRCADDR	:= ADR(vTranslation.m[3]),
				TMOUT	:= DEFAULT_ADS_TIMEOUT,
				WRITE 	:= TRUE,
				BUSY	=> ,
				ERR		=> ,
				ERRID	=> );

			State											:= 30;
		ELSE
			State											:= 90;
		END_IF

	END_IF

30: (* Roation X *)
	AdsWrite(
		TMOUT	:= DEFAULT_ADS_TIMEOUT,
		BUSY	=>,
		ERR		=>Error,
		ERRID	=>ErrorId);

	IF NOT AdsWrite.BUSY 
	THEN
		AdsWrite(WRITE:=FALSE);
		IF NOT AdsWrite.ERR 
		THEN
			AdsWrite(
				NETID	:= '',
				PORT	:= 10,
				IDXGRP	:= oidTrafo,
				IDXOFFS	:= 16#05010060,
				LEN		:= SIZEOF(VRotation.m[1]),
				SRCADDR	:= ADR(VRotation.m[1]),
				TMOUT	:= DEFAULT_ADS_TIMEOUT,
				WRITE 	:= TRUE,
				BUSY	=> ,
				ERR		=> ,
				ERRID	=> );

			State											:= 40;
		ELSE
			State											:= 90;
		END_IF
	END_IF

40: (* Roation Y *)
	AdsWrite(
		TMOUT	:= DEFAULT_ADS_TIMEOUT,
		BUSY	=>,
		ERR		=>Error,
		ERRID	=>ErrorId);

	IF NOT AdsWrite.BUSY 
	THEN
		AdsWrite(WRITE:=FALSE);
		IF NOT AdsWrite.ERR 
		THEN
			AdsWrite(
				NETID	:= '',
				PORT	:= 10,
				IDXGRP	:= oidTrafo,
				IDXOFFS	:= 16#05010061,
				LEN		:= SIZEOF(VRotation.m[2]),
				SRCADDR	:= ADR(VRotation.m[2]),
				TMOUT	:= DEFAULT_ADS_TIMEOUT,
				WRITE 	:= TRUE,
				BUSY	=> ,
				ERR		=> ,
				ERRID	=> );
			State											:= 50;
		ELSE            									
			State											:= 90;
		END_IF

	END_IF

50: (* Roation Z *)
	AdsWrite(
		TMOUT	:= DEFAULT_ADS_TIMEOUT,
		BUSY	=>,
		ERR		=>Error,
		ERRID	=>ErrorId);

	IF NOT AdsWrite.BUSY 
	THEN
		AdsWrite(WRITE:=FALSE);
		IF NOT AdsWrite.ERR 
		THEN
			AdsWrite(
				NETID	:= '',
				PORT	:= 10,
				IDXGRP	:= oidTrafo,
				IDXOFFS	:= 16#05010062,
				LEN		:= SIZEOF(VRotation.m[3]),
				SRCADDR	:= ADR(VRotation.m[3]),
				TMOUT	:= DEFAULT_ADS_TIMEOUT,
				WRITE 	:= TRUE,
				BUSY	=> ,
				ERR		=> ,
				ERRID	=> );

			State											:= 60;
		ELSE            									
			State											:= 90;
		END_IF
	END_IF

60:
	AdsWrite(
		TMOUT	:= DEFAULT_ADS_TIMEOUT,
		BUSY	=>,
		ERR		=>Error,
		ERRID	=>ErrorId);

	IF NOT AdsWrite.BUSY 
	THEN
		State												:= 90;
		AdsWrite(WRITE:=FALSE);
	END_IF

90: (* Start Lock-Param *)
	AdsWrite(
		NETID	:='',
		PORT	:= 10,
		IDXGRP	:=oidTrafo,
		IDXOFFS	:=SEL(TRUE (* Lock *), 16#05030210, 16#0503020F),
		LEN		:= 0,
		SRCADDR	:=0 ,
		WRITE	:= TRUE,
		TMOUT	:= DEFAULT_ADS_TIMEOUT,
		BUSY	=> ,
		ERR		=> ,
		ERRID	=> );

	State													:= 91;

91:
	AdsWrite(
		TMOUT	:= DEFAULT_ADS_TIMEOUT,
		BUSY	=>,
		ERR		=>,
		ERRID	=>);

	IF NOT AdsWrite.BUSY 
	THEN
		Busy 												:= FALSE;
		IF NOT AdsWrite.ERR 
		THEN
			Done											:= NOT Error;
		ELSIF NOT Error
		THEN
			Error 											:= AdsWrite.ERR;
			ErrorId 										:= AdsWrite.ERRID;
		END_IF
		IF NOT Execute 
		THEN
			State											:= 0;
		ELSE        										
			State											:= 99;
		END_IF
		AdsWrite(WRITE:=FALSE);
	END_IF

99:
	Busy 													:= FALSE;
	IF NOT Execute 
	THEN
		State												:= 0;
	END_IF

END_CASE

END_FUNCTION_BLOCK

// POUs/Motion/TF511x-KIN/03_DUTs/Positions/KIN_POSITIONS
{attribute 'no_check'}
FUNCTION_BLOCK KIN_POSITIONS 
VAR_INPUT
	Valid													:	BOOL ;
	MCS														:	KIN_POSITIONS_MCS_DUT; //Values as union
END_VAR
VAR_OUTPUT
END_VAR
VAR
END_VAR

;

METHOD PUBLIC copy : BOOL //Return value = TRUE if execution finished
VAR_IN_OUT
	Source													:	KIN_POSITIONS;
END_VAR
	Valid													:= Source.Valid;
	MCS														:= Source.MCS;
	copy													:= TRUE;
END_METHOD

METHOD PUBLIC delete : BOOL //Return value = TRUE if execution finished - Valid bit will not change
VAR_INPUT
END_VAR
	MCS.A													:= 0.0;
	MCS.B													:= 0.0;
	MCS.C													:= 0.0;
	MCS.X													:= 0.0;
	MCS.Y													:= 0.0;
	MCS.Z													:= 0.0;
	MCS.Q1													:= 0.0;
	MCS.Q2													:= 0.0;
	
	delete													:= TRUE;
END_METHOD

METHOD PUBLIC isInPos : BOOL //Return value = TRUE if axes are within window of checkPos values
VAR_IN_OUT
	CheckPos												:	KIN_POSITIONS_MCS_DUT;
	Window													:	KIN_POSITIONS_MCS_DUT;
END_VAR             										
VAR CONSTANT        										
END_VAR
IsInPos 														:= IsInPosXYZ(CheckPos,Window) AND IsInPosABC(CheckPos,Window);
END_METHOD

METHOD PUBLIC isInPosABC : BOOL //Return value = TRUE if axes are within window of checkPos values
VAR_IN_OUT
	CheckPos												:	KIN_POSITIONS_MCS_DUT;
	Window													:	KIN_POSITIONS_MCS_DUT;
END_VAR                 									
VAR CONSTANT            									
END_VAR
isInPosABC												 	:= CAM(CheckPos.A, MCS.A ,Window.A)
																AND CAM(CheckPos.B, MCS.B ,Window.B)
																AND CAM(CheckPos.C, MCS.C ,Window.C);
END_METHOD

METHOD PUBLIC isInPosByAxisNo : BOOL //Return value = TRUE selected axis is within window of checkPos values
VAR_INPUT
	No					:	INT;
END_VAR
VAR_IN_OUT
	CheckPos			:	KIN_POSITIONS_MCS_DUT;
	Window				:	KIN_POSITIONS_MCS_DUT;
END_VAR
isInPosByAxisNo													:= (CAM(CheckPos.X, MCS.X ,Window.X) OR No <> 1)
																AND (CAM(CheckPos.Y, MCS.Y ,Window.Y) OR No <> 2)
																AND (CAM(CheckPos.Z, MCS.Z ,Window.Z) OR No <> 3)
																AND (CAM(CheckPos.A, MCS.A ,Window.A) OR No <> 4)
																AND (CAM(CheckPos.B, MCS.B ,Window.B) OR No <> 5)
																AND (CAM(CheckPos.C, MCS.C ,Window.C) OR No <> 6)
																AND (CAM(CheckPos.Q1, MCS.Q1 ,Window.Q1) OR No <> 7)
																AND (CAM(CheckPos.Q2, MCS.Q2 ,Window.Q2) OR No <> 8);
END_METHOD

METHOD PUBLIC isInPosExt : BOOL //Return value = TRUE if axes are within window of checkPos values
VAR_INPUT
{attribute 'displaymode':='binary'}
	Config													:	DWORD; //Select value to be checked by bis mask .0=X or A1, .1=Y or A2, .3=Y or A3.....
END_VAR
VAR_IN_OUT
	CheckPos												:	KIN_POSITIONS_MCS_DUT;
	Window													:	KIN_POSITIONS_MCS_DUT;
END_VAR                 									
VAR CONSTANT            									
END_VAR
isInPosExt													:= (CAM(CheckPos.X, MCS.X ,Window.X) OR NOT Config.0)
																AND (CAM(CheckPos.Y, MCS.Y ,Window.Y) OR NOT Config.1)
																AND (CAM(CheckPos.Z, MCS.Z ,Window.Z) OR NOT Config.2)
																AND (CAM(CheckPos.A, MCS.A ,Window.A) OR NOT Config.3)
																AND (CAM(CheckPos.B, MCS.B ,Window.B) OR NOT Config.4)
																AND (CAM(CheckPos.C, MCS.C ,Window.C) OR NOT Config.5)
																AND (CAM(CheckPos.Q1, MCS.Q1 ,Window.Q1) OR NOT Config.6)
																AND (CAM(CheckPos.Q2, MCS.Q2 ,Window.Q2) OR NOT Config.7);
END_METHOD

METHOD PUBLIC isInPosXYZ : BOOL //Return value = TRUE if axes are within window of checkPos values
VAR_IN_OUT
	CheckPos												:	KIN_POSITIONS_MCS_DUT;
	Window													:	KIN_POSITIONS_MCS_DUT;
END_VAR                 									
VAR CONSTANT            									
END_VAR
IsInPosXYZ												 	:= CAM(CheckPos.X, MCS.X ,Window.X)
																AND CAM(CheckPos.Y, MCS.Y ,Window.Y)
																AND CAM(CheckPos.Z, MCS.Z ,Window.Z);
END_METHOD

METHOD PUBLIC reset : BOOL //Delete data and reset valid , TRUE if execution finished
VAR_INPUT
END_VAR
Delete(); 
Valid														:= FALSE;
reset														:= TRUE;
END_METHOD

END_FUNCTION_BLOCK

// POUs/Motion/TF511x-KIN/03_DUTs/Trafo/KIN_CALCTRAFO_AXPOS_PARAM
FUNCTION_BLOCK KIN_CALCTRAFO_AXPOS_PARAM
VAR_INPUT
	In														: 	ARRAY[1..8] OF LREAL;
	Out														: 	ARRAY[1..8] OF LREAL;
	MetaInfoIn												:	U_KinMetaInfo;
	MetaInfoOut												:	U_KinMetaInfo;
END_VAR
VAR_OUTPUT
END_VAR
VAR
END_VAR

METHOD delete : BOOL
VAR_INPUT
END_VAR
MEMSET(ADR(In),0,SIZEOF(In));
MEMSET(ADR(Out),0,SIZEOF(Out));
delete	:= TRUE;
END_METHOD

END_FUNCTION_BLOCK

// POUs/Motion/TF511x-KIN/03_DUTs/Trafo/KIN_STATE_OBSERVER_OID_PARAM
{attribute 'hide'}
FUNCTION_BLOCK KIN_STATE_OBSERVER_OID_PARAM
VAR_INPUT
	oid														:	UDINT := 0; (* Scara State Observer OID *)
	TooltrafoOID											:	UDINT := 0; (* ToolTrafoOID *)
	NextTrafoOID											:	UDINT := 0; (*StaticTrafoOID *)

END_VAR
VAR_OUTPUT

END_VAR
VAR
END_VAR

;

METHOD delete : BOOL
VAR_INPUT
END_VAR
	oid														:= 0;
	TooltrafoOID											:= 0;
	NextTrafoOID											:= 0;
delete	:= TRUE;
END_METHOD

END_FUNCTION_BLOCK

// POUs/Motion/TF511x-KIN/03_DUTs/Trafo/KIN_STATICTRAFO_PARAM
{attribute 'hide'}
FUNCTION_BLOCK KIN_STATICTRAFO_PARAM
VAR_INPUT
	oid														:	UDINT := 0;
	TranslationX											:	LREAL := 0.0;
	TranslationY											:	LREAL := 0.0;
	TranslationZ											:	LREAL := 0.0;
                            								
	Rotation												: LREAL := 0.0;
	RotationAxis											: INT := 2;

END_VAR
VAR_OUTPUT

END_VAR
VAR
END_VAR

;

METHOD delete : BOOL
VAR_INPUT
END_VAR
	oid														:= 0;
	TranslationX											:= 0.0;
	TranslationY											:= 0.0;
	TranslationZ											:= 0.0;
                            								
	Rotation												:= 0.0;
	RotationAxis											:= 2;
delete	:= TRUE;
END_METHOD

END_FUNCTION_BLOCK

// POUs/Motion/TF511x-KIN/03_DUTs/Trafo/KIN_TOOLTRAFO_PARAM
{attribute 'hide'}
FUNCTION_BLOCK KIN_TOOLTRAFO_PARAM
VAR_INPUT
	oid														:	UDINT := 0;
	dx														: 	LREAL := 0.0;  (* Default Tooldata at WOS *)
	dy														: 	LREAL := 0.0;  (* Default Tooldata at WOS *)
	dz														:	LREAL := 0.0;  (* Default Tooldata at WOS *)

END_VAR
VAR_OUTPUT

END_VAR
VAR
END_VAR

;

METHOD delete : BOOL
VAR_INPUT
END_VAR
	oid														:= 0;
	dx														:= 0.0;  (* Default Tooldata at WOS *)
	dy														:= 0.0;  (* Default Tooldata at WOS *)
	dz														:= 0.0;  (* Default Tooldata at WOS *)
delete	:= TRUE;
END_METHOD

END_FUNCTION_BLOCK

// POUs/Motion/TF511x-KIN/KinChannel
FUNCTION_BLOCK KinChannel EXTENDS KIN_REF
VAR_INPUT
	Admin													:	KinAdmin;
END_VAR
VAR_OUTPUT
END_VAR
VAR
END_VAR

(* Kinematic Ctrl 										*)
(********************************************************)

(* work IO ********************************************************************)
(*	IO(); *)
	
(****************************************************************************)
(* Kinematic group control													*)
(****************************************************************************)
	Admin(
		ResetTrig			:= ,
		Enable			:= ,
		Override		:= ,
		ItpChannelId	:= ,
		AxesList		:= ,
		rKINRef			:= THIS^,
		Busy			=> ,
		Done			=> ,
		Error			=> ,
		ErrorId			=> );
(****************************************************************************)

END_FUNCTION_BLOCK

// POUs/Motion/VALUE_3D
{attribute 'no_check'}
FUNCTION_BLOCK VALUE_3D
VAR_INPUT                                                            
	Valid													:	BOOL ;
	X														:	LREAL;
	Y														:	LREAL;
	Z														:	LREAL;
END_VAR
VAR_OUTPUT
END_VAR
VAR
END_VAR

;

METHOD PUBLIC copy : BOOL //Return value = TRUE if execution finished
VAR_IN_OUT
	Source													:	VALUE_3D;
END_VAR
	Valid													:= Source.Valid;
	X														:= Source.X;
	Y														:= Source.Y;
	Z														:= Source.Z;
	copy													:= TRUE;
END_METHOD

METHOD PUBLIC delete : BOOL //Return value = TRUE if execution finished - Valid bit will not change
VAR_INPUT
END_VAR
	X					 									:= 0.0;	
	Y					 									:= 0.0;	
	Z					 									:= 0.0;	
	delete													:= TRUE;
END_METHOD

METHOD PUBLIC InPos : BOOL //Return value = TRUE axes is within window of checkPos values
VAR_IN_OUT
	CheckPos												:	VALUE_3D;
	Window													:	VALUE_3D;
END_VAR
InPos														:= CAM(CheckPos.X, X ,Window.X)
																AND CAM(CheckPos.Y, Y ,Window.Y)
																AND CAM(CheckPos.Z, Z ,Window.Z);
END_METHOD

METHOD PUBLIC InPosByAxisNo : BOOL //Return value = TRUE selected axis is within window of checkPos values
VAR_INPUT
	No					:	INT;
END_VAR
VAR_IN_OUT
	CheckPos			:	VALUE_3D;
	Window				:	VALUE_3D;
END_VAR
InPosByAxisNo													:= (CAM(CheckPos.X, X ,Window.X) OR No <> 1)
																AND (CAM(CheckPos.Y, Y ,Window.Y) OR No <> 2)
																AND (CAM(CheckPos.Z, Z ,Window.Z) OR No <> 3);
END_METHOD

METHOD PUBLIC InPosXY : BOOL //Return value = TRUE if axes are within window of checkPos values
VAR_IN_OUT
	CheckPos			:	VALUE_3D;
	Window				:	VALUE_3D;
END_VAR
InPosXY 													:= CAM(CheckPos.X, X ,Window.X)
																AND CAM(CheckPos.Y, Y ,Window.Y);
END_METHOD

METHOD PUBLIC InPosXZ : BOOL //Return value = TRUE if axes are within window of checkPos values
VAR_IN_OUT
	CheckPos			:	VALUE_3D;
	Window				:	VALUE_3D;
	
END_VAR
InPosXZ														:= CAM(CheckPos.X, X ,Window.X)
																AND CAM(CheckPos.Z, Z ,Window.Z);
END_METHOD

METHOD PUBLIC InPosYZ : BOOL //Return value = TRUE if axes are within window of checkPos values
VAR_IN_OUT
	CheckPos			:	VALUE_3D;
	Window				:	VALUE_3D;
	
END_VAR
InPosYZ													:= CAM(CheckPos.Y, Y ,Window.Y)
																AND CAM(CheckPos.Z, Z ,Window.Z);
END_METHOD

METHOD PUBLIC reset : BOOL //Delete data and reset valid , TRUE if execution finished
VAR_INPUT
END_VAR
Delete();
Valid														:= FALSE;
reset														:= TRUE;
END_METHOD

END_FUNCTION_BLOCK

// POUs/Motion/VALUE_6D
{attribute 'no_check'}
FUNCTION_BLOCK VALUE_6D 
VAR_INPUT
	Valid													:	BOOL ;
	X														:	LREAL;
	Y														:	LREAL;
	Z														:	LREAL;
	A														:		LREAL; //Rx
	B														:		LREAL; //Ry
	C														:		LREAL; //Rz	
END_VAR
VAR_OUTPUT
END_VAR
VAR
END_VAR

;

METHOD PUBLIC copy : BOOL //Return value = TRUE if execution finished
VAR_IN_OUT
	Source													:	VALUE_6D;
END_VAR
	Valid													:= Source.Valid;
	X														:= Source.X;
	Y														:= Source.Y;
	Z														:= Source.Z;
	A														:= Source.A;
	B														:= Source.B;
	C														:= Source.C;
	copy													:= TRUE;
END_METHOD

METHOD PUBLIC delete : BOOL //Return value = TRUE if execution finished - Valid bit will not change
VAR_INPUT
END_VAR
	X					 									:= 0.0;	
	Y					 									:= 0.0;	
	Z					 									:= 0.0;	
	A						 								:= 0.0;	
	B						 								:= 0.0;	
	C						 								:= 0.0;	
	delete													:= TRUE;
END_METHOD

METHOD PUBLIC inPos : BOOL //Return value = TRUE if axes are within window of checkPos values
VAR_IN_OUT
	CheckPos												:	VALUE_6D;
	Window													:	VALUE_6D;
END_VAR             										
VAR CONSTANT        										
END_VAR
InPos 														:= CAM(CheckPos.X, X, Window.X)
																AND CAM(CheckPos.Y, Y ,Window.Y)
																AND CAM(CheckPos.Z, Z,Window.Z)
																AND CAM(CheckPos.A, A, Window.A)
																AND CAM(CheckPos.B, B ,Window.B)
																AND CAM(CheckPos.C, C,Window.C);
END_METHOD

METHOD PUBLIC InPosABC : BOOL //Return value = TRUE if axes are within window of checkPos values
VAR_IN_OUT
	CheckPos												:	VALUE_6D;
	Window													:	VALUE_6D;
END_VAR                 									
VAR CONSTANT            									
END_VAR
InPosABC												 	:= CAM(CheckPos.A, A ,Window.A)
																AND CAM(CheckPos.B, B ,Window.B)
																AND CAM(CheckPos.C, C ,Window.C);
END_METHOD

METHOD PUBLIC InPosAC : BOOL //Return value = TRUE if axes are within window of checkPos values
VAR_IN_OUT
	CheckPos												:	VALUE_6D;
	Window													:	VALUE_6D;
END_VAR                 									
VAR CONSTANT            									
END_VAR
InPosAC													 	:= CAM(CheckPos.A, A ,Window.A)
																AND CAM(CheckPos.C, C ,Window.C);
END_METHOD

METHOD PUBLIC inPosByAxisNo : BOOL //Return value = TRUE selected axis is within window of checkPos values
VAR_INPUT
	No					:	INT;
END_VAR
VAR_IN_OUT
	CheckPos			:	VALUE_6D;
	Window				:	VALUE_6D;
END_VAR
inPosByAxisNo													:= (CAM(CheckPos.X, X ,Window.X) OR No <> 1)
																AND (CAM(CheckPos.Y, Y ,Window.Y) OR No <> 2)
																AND (CAM(CheckPos.Z, Z ,Window.Z) OR No <> 3)
																AND (CAM(CheckPos.A, A ,Window.A) OR No <> 4)
																AND (CAM(CheckPos.B, B ,Window.B) OR No <> 5)
																AND (CAM(CheckPos.C, C ,Window.C) OR No <> 6);
END_METHOD

METHOD PUBLIC inPosXY : BOOL //Return value = TRUE if axes are within window of checkPos values
VAR_IN_OUT
	CheckPos												:	VALUE_6D;
	Window													:	VALUE_6D;
END_VAR                 									
VAR CONSTANT            									
END_VAR
InPosXY													 	:= CAM(CheckPos.X, X ,Window.X)
																AND CAM(CheckPos.Y, Y ,Window.Y);
END_METHOD

METHOD PUBLIC InPosXYZ : BOOL //Return value = TRUE if axes are within window of checkPos values
VAR_IN_OUT
	CheckPos												:	VALUE_6D;
	Window													:	VALUE_6D;
END_VAR                 									
VAR CONSTANT            									
END_VAR
InPosXYZ												 	:= CAM(CheckPos.X, X ,Window.X)
																AND CAM(CheckPos.Y, Y ,Window.Y)
																AND CAM(CheckPos.Z, Z ,Window.Z);
END_METHOD

METHOD PUBLIC inPosXZ : BOOL //Return value = TRUE if axes are within window of checkPos values
VAR_IN_OUT
	CheckPos												:	VALUE_6D;
	Window													:	VALUE_6D;
END_VAR                 									
VAR CONSTANT            									
END_VAR
InPosXZ												 	:= CAM(CheckPos.X, X ,Window.X)
																AND CAM(CheckPos.Z, Z ,Window.Z);
END_METHOD

METHOD PUBLIC inPosYZ : BOOL //Return value = TRUE if axes are within window of checkPos values
VAR_IN_OUT
	CheckPos												:	VALUE_6D;
	Window													:	VALUE_6D;
END_VAR                 									
VAR CONSTANT            									
END_VAR
InPosYZ													 	:= CAM(CheckPos.Y, Y ,Window.Y)
																AND CAM(CheckPos.Z, Z ,Window.Z);
END_METHOD

METHOD PUBLIC reset : BOOL //Delete data and reset valid , TRUE if execution finished
VAR_INPUT
END_VAR
Delete(); 
Valid														:= FALSE;
reset														:= TRUE;
END_METHOD

END_FUNCTION_BLOCK

// POUs/Safety/Diag/SafetyIODeviceDiag_wEvents
{attribute 'no_check'}
FUNCTION_BLOCK SafetyIODeviceDiag_wEvents
VAR CONSTANT
	MIN_EVENT												:	INT := 1;
	MAX_EVENT												:	INT := 10;
	
//Event conn diag code xxxx					| FB1 - Msg 1..15
//Event conn diag code .4 					| FB2 - Msg 16
//Event conn diag code .5 					| FB3 - Msg 17
                                        	
//Event internal error 						| FB1 - Msg 18
                                        	
//Event send TextId 						| FB4 - Msg 19
                                        	
//Event send AX5xxx Err Chn 1 				| FB5 - Msg 20
//Event send AX5xxx Err Chn 1 				| FB6 - Msg 21
                                        	
//Event send Ex19 Err Debug 0x800E:0A 		| FB4 - Msg 22
//Event send Ex19 Err Debug 0x800E:0B		| FB5 - Msg 23
//Event send Ex19 Err Debug 0x800E:0C 		| FB6 - Msg 24
//Event send Ex19 Err Debug 0x800E:0D 		| FB7 - Msg 25
//Event send Ex19 Err Debug 0x800E:13 		| FB8 - Msg 26
//Event send Ex19 Err Debug 0x800E:14 		| FB9 - Msg 27
//Event send Ex19 Err Debug 0x800E:15		| FB10- Msg 28
                                        	
//Event send EL29 Err Debug 0x800E:0C 		| FB4 - Msg 30 (Querschluss bit 0..3)
//Event send EL29 Err Debug 0x800E:0C 		| FB4 - Msg 31 (Open load bit 4..7)
//Event send EL29 Err Debug 0x800E:0D		| FB5 - Msg 32
//Event send EL29 Err Debug 0x800E:0E 		| FB6 - Msg 33
//Event send EL29 Err Debug 0x800E:0E 		| FB7 - Msg 34
//Event send EL29 Err Debug 0x800E:0E 		| FB8 - Msg 35

                                        	
//Event send EK19 Err Debug 0x800E:0A		| FB4 - Msg 22 
//Event send EK19 Err Debug 0x800E:0B		| FB5 - Msg 23 
//Event send EK19 Err Debug 0x800E:0C 		| FB6 - Msg 24 
//Event send EK19 Err Debug 0x800E:0D 		| FB7 - Msg 25 
//Event send EK19 Err Debug 0x800E:0E	 	| FB8 - Msg 36..45
END_VAR
VAR_INPUT
	Enable													:	BOOL;	//FB will be processed as long as enable is TRUE 
	ConfirmTrig												:	BOOL;	//Resets error with rising edge 
	SourceId												:	UDINT;	//Multisource id 
	EcMasterDevId											:	UINT;	//Map to EtherCAT Master DevId
END_VAR                 									
VAR_OUTPUT              									
	Connected												:	BOOL;
	{attribute 'displaymode':='binary'}
	Status													:	DWORD;	//current status of event
	NoOfActiveEvents										:	INT;
END_VAR                 									

VAR(* internal *)
	state													:	INT := 0;
	{attribute 'displaymode':='binary'}
	ConnMsgDiagCode											:	BYTE;
	Read													:	SafetyIODeviceDiagRead;
   	Event													:	ARRAY [MIN_EVENT..MAX_EVENT] OF EventHandling; 
	DevTypeAndAddr											:	STRING(30);
    DebugData												:	 word;                 								                            	
	i														:	INT;
END_VAR

(* Safety IO device diag with events		V2	*)
(************************************************)

(* Status connected ***************************************************)
	Connected 												:= Read.AdsAddr.port <> 0;
	
(* Read adress and type ***********************************************)
	IF Enable AND Connected AND Read.MsgInfoDiag <> 0 OR State <> 0
	THEN
		CASE State OF
		0:	
			IF Read.MsgInfoDiag <> 0
			THEN
				Read(Execute := FALSE);
				Read(Execute := TRUE, EcMasterDevId := EcMasterDevId);
				State										:= State + 1;
			END_IF
			
		1: //Read diag data from device
			Read(Execute := TRUE, EcMasterDevId := EcMasterDevId);
			IF NOT Read.Busy
			THEN
	
				IF Read.Error
				THEN
					Event[1].Text1							:= SEL(Read.Name = '',Read.Name , '<ERR_READ_DIAG>');
					DevTypeAndAddr							:= SEL(Read.DevType = '', Read.DevType, '<Unknown>');
					DevTypeAndAddr							:= CONCAT(DevTypeAndAddr, CONCAT(' (Ec Addr.', CONCAT(TO_STRING(Read.AdsAddr.port),')')));	
					Event[1].Text2							:= CONCAT(' - ErrorID ', DWORD_TO_HEXSTR(TO_DWORD(Read.ErrorID),4,FALSE));
					Event[1].Text2							:= CONCAT(Event[1].Text2 , CONCAT(' in state ', TO_STRING(Read.DiagMsgTextId)));
					Event[1].SourceId						:= SourceId;
					Event[1].Flag							:= TRUE;
					State									:= 98;
				ELSIF Event[1].SourceId = 0
				THEN //Init device information 
					FOR i := MIN_EVENT TO MAX_EVENT
					DO
						Event[i].Text1						:= Read.Name;
						DevTypeAndAddr						:= CONCAT(Read.DevType, ' (FSOE Addr.');
						DevTypeAndAddr						:= CONCAT(DevTypeAndAddr, CONCAT(TO_STRING(Read.FSOEAddr), ')'));	
						Event[i].SourceId					:= SourceId;
					END_FOR
					State									:= 99;
				ELSE
					State									:= 99;
				END_IF		
				Read(Execute := FALSE);
			END_IF
			
		98: //Show internal error
			Event[1](
				Flag	:= Event[1].Flag AND NOT Event[1].ConfirmTrig,
				ConfirmTrig:= ConfirmTrig OR Read.MsgInfoDiag = 0, 
				MsgId	:= 18, 
				pText3	:= ADR(DevTypeAndAddr),
				Status	=> Status);	
			IF NOT Event[1].Status.31 
			THEN
				NoOfActiveEvents							:= 0;
				state										:= 0;
			ELSE
				NoOfActiveEvents							:= 1;
			END_IF
			
		99: //Fire events
			IF Read.MsgInfoDiag = 0 AND NOT Status.31
			THEN //Go back to 0 if messages cleared
				State 										:= 0;
			ELSE
				//Show connection error events
				_eventsConnDiag();
				
				//Fire device events
				IF Read.pDebugData <> 0 
				THEN //Safety devices without diag history object
					IF Read.DebugDataMaxId = 16#08 AND_THEN FIND(Read.DevType, 'AX580') <> 0
					THEN
						_eventsAX580x(Read.MsgInfoDiag <> 0);
					ELSIF Read.DebugDataMaxId = 16#10 AND_THEN Read.DevType = 'EL2904'
					THEN
						_eventsEL2904(Read.MsgInfoDiag <> 0);
					ELSIF Read.DebugDataMaxId = 16#40 AND_THEN Read.DevType = 'EK1914' 
					THEN
						_eventsEK1914(Read.MsgInfoDiag <> 0);
					ELSIF Read.DebugDataMaxId >= 16#10 
					THEN//EL1904 or EP1908
						_eventsEx190x(Read.MsgInfoDiag <> 0);		
					ELSE //Show internal error 
						Event[4](
							Flag	:= Read.MsgInfoDiag <> 0,
							ConfirmTrig:= ConfirmTrig OR Read.MsgInfoDiag = 0, 
							MsgId	:= 18, 
							Text2	:= CONCAT(' Invalid lenght of Coe object 0x800E for device ', TO_STRING(Read.DebugDataMaxId)),
							pText3	:= ADR(DevTypeAndAddr));	
					END_IF
				ELSE //TwinSAFE terminal with diag history  
					_eventsDiagHistory(Read.MsgInfoDiag <> 0);
				END_IF			
			END_IF		
						   	
			//Check whether one event is active **************************************
			NoOfActiveEvents 		 						:= 0;			
			Status											:= 0;						
			FOR i := MIN_EVENT TO MAX_EVENT
			DO 
				IF Event[i].Status.31 THEN NoOfActiveEvents := NoOfActiveEvents + 1 ; END_IF
				Status										:= Status OR Event[i].Status;
			END_FOR
		END_CASE
	END_IF

(*******************************************************************************)

METHOD PRIVATE _eventsAX580x : BOOL
VAR_INPUT
	ShowEvent										:	BOOL;
END_VAR
(* Fire AX5000 events ***********************************)
	//Send AX58xx diag code channel 1 
	IF Read.pDebugData^[1] = 0
	THEN
		Event[5].Text2										:= CONCAT('0x',DWORD_TO_HEXSTR(TO_DWORD(Read.pDebugData^[7]),4,FALSE));
	ELSE
		Event[5].Text2										:= '<Set CoE object 0xFA10:01 = 0>';
	END_IF
 
	Event[5](
		Flag	:= ShowEvent AND Read.msgSevyIsError ,
		ConfirmTrig:= ConfirmTrig, 
		MsgId	:= 20, 
		Class	:= ,
		pText3	:= ADR(DevTypeAndAddr));	
		
	//Send AX58xx diag code channel 2
	IF Read.pDebugData^[1] = 0
	THEN
		Event[6].Text2										:= CONCAT('0x',DWORD_TO_HEXSTR(TO_DWORD(Read.pDebugData^[8]),4,FALSE));
	ELSE
		Event[6].Text2										:=  '<Set CoE object 0xFA10:01 = 0>';
	END_IF
 
	Event[6](
		Flag	:= ShowEvent AND Read.msgSevyIsError ,
		ConfirmTrig:= ConfirmTrig, 
		MsgId	:= 21, 
		Class	:= ,
		pText3	:= ADR(Read.Name));

(******************************************************)
END_METHOD

METHOD PRIVATE _eventsConnDiag : BOOL
VAR_INPUT
END_VAR
(* Fire event for connection error code ************************************)
	ConnMsgDiagCode											:= 16#0F AND Read.MsgInfoDiag; 
	IF ConnMsgDiagCode <> 0 OR Event[1].Status.31
	THEN
		Event[1](
			Flag	:= ConnMsgDiagCode <> 0 AND NOT (ConnMsgDiagCode = 2#1101 AND Read.MsgInfoDiag.5),
			ConfirmTrig:= ConfirmTrig, 
			MsgId	:= ConnMsgDiagCode,  //1..15 		
			pText3	:= ADR(DevTypeAndAddr));	
	END_IF
	
	//Fire event xxx1 xxxx FSoE Slave error detected
	IF Read.MsgInfoDiag.4 OR Event[2].Status.31
	THEN
		Event[2](
			Flag	:= Read.MsgInfoDiag.4,
			ConfirmTrig:= ConfirmTrig, 
			MsgId	:= 16,		
			pText3	:= ADR(DevTypeAndAddr));	
	END_IF

(*
	//Fire event xx1x xxxx FSoE Slave notifies Failsafe Value active
	IF Read.MsgInfoDiag.5 OR Event[3].Status.31
	THEN
		Event[3](
			Flag	:= Read.MsgInfoDiag.5,
			ConfirmTrig:= ConfirmTrig, 
			MsgId	:= 17,		
			pText3	:= ADR(DevTypeAndAddr));		
	END_IF
*)	
	(*
	Tabelle 2-4: Diagnose-Informationen einer Connection
	Wert Beschreibung
	xxxx 0001 invalid command
	xxxx 0010 unknown command
	xxxx 0011 invalid connection ID
	xxxx 0100 invalid CRC
	xxxx 0101 Watchdog run out of time
	xxxx 0110 invalid FSoE-Adress
	xxxx 0111 invalid data
	xxxx 1000 invalid length of communicatoin parameter Kommunikationsparameterlänge
	xxxx 1001 invalid communicatoin parameter
	xxxx 1010 invalid operator parameter length
	xxxx 1011 invalid operator parameter
	xxxx 1100 FSoE Master Reset
	xxxx 1101 Module fault on slave detected with activated option "Modulfault is ComError"
	xxxx 1110 Module fault on EL290x at activated with option "Error achnowledge active"
	xxxx 1111 Slave not started or unexpected error argument
	
	*)
		
(***********************************************************************)
END_METHOD

METHOD PRIVATE _eventsDiagHistory : BOOL
VAR_INPUT
	ShowEvent										:	BOOL;
END_VAR
(* Send diag message textId ********************************************)
	Event[4](
		Flag	:= ShowEvent AND Read.msgSevyIsError ,
		ConfirmTrig:= ConfirmTrig, 
		MsgId	:= 19, 
		Text2	:= CONCAT('0x',DWORD_TO_HEXSTR(TO_DWORD(Read.DiagMsgTextId),4,FALSE)),
		pText3	:= ADR(DevTypeAndAddr));

(******************************************************)
END_METHOD

METHOD PRIVATE _eventsEK1914 : BOOL
VAR_INPUT
	ShowEvent										:	BOOL;
END_VAR
// Fire events for of EK1914 ****************************************)

		(* error during sensor-test *)
		Event[4].Flag 										:= Read.pDebugData^[16#0A] <> 0;
		IF Event[4].Flag OR Event[4].Status.31
		THEN
			DebugData										:= Read.pDebugData^[16#0A];
			Event[4].Text2									:= '';
			IF DebugData.0 THEN Event[4].Text2 				:= CONCAT(Event[4].Text2, '|1'); END_IF
			IF DebugData.1 THEN Event[4].Text2 				:= CONCAT(Event[4].Text2, '|2'); END_IF
		(*	IF DebugData.2 THEN Event[4].Text2 				:= CONCAT(Event[4].Text2, '|3'); END_IF
			IF DebugData.3 THEN Event[4].Text2 				:= CONCAT(Event[4].Text2, '|4');  END_IF
			IF DebugData.4 THEN Event[4].Text2 				:= CONCAT(Event[4].Text2, '|5'); END_IF
			IF DebugData.5 THEN Event[4].Text2 				:= CONCAT(Event[4].Text2, '|6'); END_IF
			IF DebugData.6 THEN Event[4].Text2 				:= CONCAT(Event[4].Text2, '|7'); END_IF
			IF DebugData.7 THEN Event[4].Text2 				:= CONCAT(Event[4].Text2, '|8');  END_IF *)
			Event[4].Text2 									:= CONCAT(Event[4].Text2, '|'); 			
			
			Event[4](
				Flag	:= ShowEvent ,
				ConfirmTrig:= ConfirmTrig, 
				MsgId	:= 22, 
				pText3	:= ADR(DevTypeAndAddr))	;
		END_IF

		(* Zweikanalauswertung fehlerhaft *)
		Event[5].Flag 										:= Read.pDebugData^[16#0B] <> 0;
		IF Event[5].Flag OR Event[5].Status.31
		THEN
			DebugData										:= Read.pDebugData^[16#0B];
			Event[5].Text2									:= '';
			IF DebugData.0 THEN Event[5].Text2 				:= CONCAT(Event[5].Text2, '|1+2'); END_IF
		(*	IF DebugData.1 THEN Event[5].Text2 				:= CONCAT(Event[5].Text2, '|3+4'); END_IF
			IF DebugData.2 THEN Event[5].Text2 				:= CONCAT(Event[5].Text2, '|5+6'); END_IF
			IF DebugData.3 THEN Event[5].Text2 				:= CONCAT(Event[5].Text2, '|7+8');  END_IF *)
			Event[5].Text2 									:= CONCAT(Event[5].Text2, '|'); 
			
			Event[5](
				Flag	:= ShowEvent ,
				ConfirmTrig:= ConfirmTrig, 
				MsgId	:= 23, 
				pText3	:= ADR(DevTypeAndAddr))	;
		END_IF

		(* Fehler Eingangspaar Trittmattenbetriebsart - Eingangspaar uneinig *)
		Event[6].Flag 										:= Read.pDebugData^[16#0C] <> 0;
		IF Event[6].Flag OR Event[6].Status.31
		THEN
			DebugData										:= Read.pDebugData^[16#0C];
			Event[6].Text2									:= '';
			IF DebugData.0 THEN Event[6].Text2 				:= CONCAT(Event[6].Text2, '|1+2'); END_IF
		(*	IF DebugData.1 THEN Event[6].Text2 				:= CONCAT(Event[6].Text2, '|3+4'); END_IF
			IF DebugData.2 THEN Event[6].Text2 				:= CONCAT(Event[6].Text2, '|5+6'); END_IF
			IF DebugData.3 THEN Event[6].Text2 				:= CONCAT(Event[6].Text2, '|7+8');  END_IF *)
			Event[6].Text2 									:= CONCAT(Event[6].Text2, '|'); 
			
			Event[6](
				Flag	:= ShowEvent ,
				ConfirmTrig:= ConfirmTrig, 
				MsgId	:= 24, 
				pText3	:= ADR(DevTypeAndAddr))	;
		END_IF

		(* Fehler Trittmattenbetriebsart Fremdeinspeisung *)
		Event[7].Flag 										:= Read.pDebugData^[16#0D] <> 0;
		IF Event[7].Flag OR Event[7].Status.31
		THEN
			DebugData										:= Read.pDebugData^[16#0D];
			Event[7].Text2									:= '';
			IF DebugData.0 THEN Event[7].Text2 				:= CONCAT(Event[7].Text2, '|1'); END_IF
			IF DebugData.1 THEN Event[7].Text2 				:= CONCAT(Event[7].Text2, '|2'); END_IF
		(*	IF DebugData.2 THEN Event[7].Text2 				:= CONCAT(Event[7].Text2, '|3'); END_IF
			IF DebugData.3 THEN Event[7].Text2 				:= CONCAT(Event[7].Text2, '|4');  END_IF
			IF DebugData.4 THEN Event[7].Text2 				:= CONCAT(Event[7].Text2, '|5'); END_IF
			IF DebugData.5 THEN Event[7].Text2 				:= CONCAT(Event[7].Text2, '|6'); END_IF
			IF DebugData.6 THEN Event[7].Text2 				:= CONCAT(Event[7].Text2, '|7'); END_IF
			IF DebugData.7 THEN Event[7].Text2 				:= CONCAT(Event[7].Text2, '|8');  END_IF *)
			Event[7].Text2 									:= CONCAT(Event[7].Text2, '|'); 
			
			Event[7](
				Flag	:= ShowEvent ,
				ConfirmTrig:= ConfirmTrig, 
				MsgId	:= 25, 
				pText3	:= ADR(DevTypeAndAddr))	;
		END_IF
		
		(* Fehler Ausgänge *)
		IF Read.pDebugData^[16#0E] <> 0 OR Event[8].Status.31 
		THEN
			DebugData										:= Read.pDebugData^[16#0E];
			
			CASE DebugData OF
			5:		Event[8].MsgId							:= 36;
			6:		Event[8].MsgId							:= 37;
			10:		Event[8].MsgId							:= 38;
			11:		Event[8].MsgId							:= 39;
			21..27:	Event[8].MsgId							:= 40;
			30..33:	Event[8].MsgId							:= 41;
			101:	Event[8].MsgId							:= 42;
			102:	Event[8].MsgId							:= 43;
			103:	Event[8].MsgId							:= 44;
			104:	Event[8].MsgId							:= 45;
			ELSE
				Event[8].MsgId								:= 0;
			END_CASE
				
			Event[8](
				Flag	:= ShowEvent AND Event[8].MsgId <> 0 ,
				ConfirmTrig:= ConfirmTrig, 
				MsgId	:= , 
				pText3	:= ADR(DevTypeAndAddr))	;
				
		END_IF		
(********************************************************************************)
END_METHOD

METHOD PRIVATE _eventsEL2904 : BOOL
VAR_INPUT
	ShowEvent										:	BOOL;
END_VAR
// Fire events for EL2904

	(* Fremeinspeisung oder Querschluss *)
	Event[4].Flag 										:= (Read.pDebugData^[16#0C] AND 16#000F) <> 0;
	IF Event[4].Flag OR Event[4].Status.31
	THEN
		DebugData										:= Read.pDebugData^[16#0C];
		Event[4].Text2									:= '';
		IF DebugData.0 THEN Event[4].Text2 				:= CONCAT(Event[4].Text2, '|1'); END_IF
		IF DebugData.1 THEN Event[4].Text2 				:= CONCAT(Event[4].Text2, '|2'); END_IF
		IF DebugData.2 THEN Event[4].Text2 				:= CONCAT(Event[4].Text2, '|3'); END_IF
		IF DebugData.3 THEN Event[4].Text2 				:= CONCAT(Event[4].Text2, '|4');  END_IF
		Event[4].Text2 									:= CONCAT(Event[4].Text2, '|'); 
			
		Event[4](
			Flag	:= ShowEvent ,
			ConfirmTrig:= ConfirmTrig, 
			MsgId	:= 30, 
			pText3	:= ADR(DevTypeAndAddr))	;
	END_IF

	(* Open load oder Mindeststrom (20mA) unterschritten, oder Maximalstrom ueberschritten (500mA) *)
	Event[5].Flag 										:= (Read.pDebugData^[16#0C] AND 16#00F0) <> 0;
	IF Event[5].Flag OR Event[5].Status.31
	THEN
		DebugData										:= Read.pDebugData^[16#0C];
		Event[5].Text2									:= '';
		IF DebugData.4 THEN Event[5].Text2 				:= CONCAT(Event[5].Text2, '|1'); END_IF
		IF DebugData.5 THEN Event[5].Text2 				:= CONCAT(Event[5].Text2, '|2'); END_IF
		IF DebugData.6 THEN Event[5].Text2 				:= CONCAT(Event[5].Text2, '|3'); END_IF
		IF DebugData.7 THEN Event[5].Text2 				:= CONCAT(Event[5].Text2, '|4');  END_IF
		Event[5].Text2 									:= CONCAT(Event[5].Text2, '|'); 
		
		Event[5](
			Flag	:= ShowEvent ,
			ConfirmTrig:= ConfirmTrig, 
			MsgId	:= 31, 
			pText3	:= ADR(DevTypeAndAddr));	
	END_IF
	
	(* Fehler Feldspannung Power Kontakte *)
	Event[6].Flag 										:= Read.pDebugData^[16#0D] <> 0;
	IF Event[6].Flag OR Event[6].Status.31
	THEN
		DebugData										:= Read.pDebugData^[16#0D];
		Event[6].Text2									:= '';
		IF DebugData.0 THEN 
			Event[6].Text2 								:= CONCAT(Event[6].Text2, '|Y'); 
		ELSE                                                                       
			Event[6].Text2 								:= CONCAT(Event[6].Text2, '|N'); 
		END_IF                                                                     
		IF DebugData.1 THEN                                                        
			Event[6].Text2 								:= CONCAT(Event[6].Text2, '|Y'); 
		ELSE                                                                       
			Event[6].Text2 								:= CONCAT(Event[6].Text2, '|N'); 
		END_IF
		Event[6].Text2 									:= CONCAT(Event[6].Text2, '|'); 
		
		Event[6](
			Flag	:= ShowEvent ,
			ConfirmTrig:= ConfirmTrig, 
			MsgId	:= 32, 
			pText3	:= ADR(DevTypeAndAddr))	;
	END_IF
	
	(* Temperaturfehler *)
	IF Read.pDebugData^[16#0E] <> 0 OR Event[7].Status.31 OR Event[8].Status.31 OR Event[9].Status.31
	THEN
		DebugData										:= Read.pDebugData^[16#0E];
		
		//Uebertemperatur
		Event[7](
			Flag	:= ShowEvent AND(DebugData.0 OR DebugData.1 OR DebugData.2),
			ConfirmTrig:= ConfirmTrig, 
			MsgId	:= 33, 
			pText3	:= ADR(DevTypeAndAddr));	
			
		//Untertemperatur
		Event[8](
			Flag	:= ShowEvent AND(DebugData.3 OR DebugData.4 OR DebugData.5),
			ConfirmTrig:= ConfirmTrig, 
			MsgId	:= 34, 
			pText3	:= ADR(DevTypeAndAddr))	;
			
		//Temp. Differenz
		Event[9](
			Flag	:= ShowEvent AND(DebugData.6 OR DebugData.6),
			ConfirmTrig:= ConfirmTrig, 
			MsgId	:= 35, 
			pText3	:= ADR(DevTypeAndAddr))	;
	END_IF
		
(***********************************************************************)
END_METHOD

METHOD PRIVATE _eventsEx190x : BOOL
VAR_INPUT
	ShowEvent										:	BOOL;
END_VAR
VAR
	DebugData												:	WORD;
END_VAR
// Fire events for EL1904 and EP1908 errors

	(* error during sensor-test *)
	Event[4].Flag 										:= Read.pDebugData^[16#0A] <> 0;
	IF Event[4].Flag OR Event[4].Status.31
	THEN
		DebugData										:= Read.pDebugData^[16#0A];
		Event[4].Text2									:= '';
		IF DebugData.0 THEN Event[4].Text2 				:= CONCAT(Event[4].Text2, '|1'); END_IF
		IF DebugData.1 THEN Event[4].Text2 				:= CONCAT(Event[4].Text2, '|2'); END_IF
		IF DebugData.2 THEN Event[4].Text2 				:= CONCAT(Event[4].Text2, '|3'); END_IF
		IF DebugData.3 THEN Event[4].Text2 				:= CONCAT(Event[4].Text2, '|4');  END_IF
		IF DebugData.4 THEN Event[4].Text2 				:= CONCAT(Event[4].Text2, '|5'); END_IF
		IF DebugData.5 THEN Event[4].Text2 				:= CONCAT(Event[4].Text2, '|6'); END_IF
		IF DebugData.6 THEN Event[4].Text2 				:= CONCAT(Event[4].Text2, '|7'); END_IF
		IF DebugData.7 THEN Event[4].Text2 				:= CONCAT(Event[4].Text2, '|8');  END_IF
		Event[4].Text2 									:= CONCAT(Event[4].Text2, '|'); 
		
		Event[4](
			Flag	:= ShowEvent ,
			ConfirmTrig:= ConfirmTrig, 
			MsgId	:= 22, 
			pText3	:= ADR(DevTypeAndAddr))	;
	END_IF

	(* Zweikanalauswertung fehlerhaft *)
	Event[5].Flag 										:= Read.pDebugData^[16#0B] <> 0;
	IF Event[5].Flag OR Event[5].Status.31
	THEN
		DebugData										:= Read.pDebugData^[16#0B];
		Event[5].Text2									:= '';
		IF DebugData.0 THEN Event[5].Text2 				:= CONCAT(Event[5].Text2, '|1+2'); END_IF
		IF DebugData.1 THEN Event[5].Text2 				:= CONCAT(Event[5].Text2, '|3+4'); END_IF
		IF DebugData.2 THEN Event[5].Text2 				:= CONCAT(Event[5].Text2, '|5+6'); END_IF
		IF DebugData.3 THEN Event[5].Text2 				:= CONCAT(Event[5].Text2, '|7+8');  END_IF
		Event[5].Text2 									:= CONCAT(Event[5].Text2, '|'); 		
	
		Event[5](
			Flag	:= ShowEvent ,
			ConfirmTrig:= ConfirmTrig, 
			MsgId	:= 23, 
			pText3	:= ADR(DevTypeAndAddr))	;
	END_IF

	(* Fehler Eingangspaar Trittmattenbetriebsart - Eingangspaar uneinig *)
	Event[6].Flag 										:= Read.pDebugData^[16#0C] <> 0;
	IF Event[6].Flag OR Event[6].Status.31
	THEN
		DebugData										:= Read.pDebugData^[16#0C];
		Event[6].Text2									:= '';
		IF DebugData.0 THEN Event[6].Text2 				:= CONCAT(Event[6].Text2, '|1+2'); END_IF
		IF DebugData.1 THEN Event[6].Text2 				:= CONCAT(Event[6].Text2, '|3+4'); END_IF
		IF DebugData.2 THEN Event[6].Text2 				:= CONCAT(Event[6].Text2, '|5+6'); END_IF
		IF DebugData.3 THEN Event[6].Text2 				:= CONCAT(Event[6].Text2, '|7+8');  END_IF
		Event[6].Text2 									:= CONCAT(Event[6].Text2, '|'); 
				
		Event[6](
			Flag	:= ShowEvent ,
			ConfirmTrig:= ConfirmTrig, 
			MsgId	:= 24, 
			pText3	:= ADR(DevTypeAndAddr))	;
	END_IF

	(* Fehler Trittmattenbetriebsart Fremdeinspeisung *)
	Event[7].Flag 										:= Read.pDebugData^[16#0D] <> 0;
	IF Event[7].Flag OR Event[7].Status.31
	THEN
		DebugData										:= Read.pDebugData^[16#0D];
		Event[7].Text2									:= '';
		IF DebugData.0 THEN Event[7].Text2 				:= CONCAT(Event[7].Text2, '|1'); END_IF
		IF DebugData.1 THEN Event[7].Text2 				:= CONCAT(Event[7].Text2, '|2'); END_IF
		IF DebugData.2 THEN Event[7].Text2 				:= CONCAT(Event[7].Text2, '|3'); END_IF
		IF DebugData.3 THEN Event[7].Text2 				:= CONCAT(Event[7].Text2, '|4');  END_IF
		IF DebugData.4 THEN Event[7].Text2 				:= CONCAT(Event[7].Text2, '|5'); END_IF
		IF DebugData.5 THEN Event[7].Text2 				:= CONCAT(Event[7].Text2, '|6'); END_IF
		IF DebugData.6 THEN Event[7].Text2 				:= CONCAT(Event[7].Text2, '|7'); END_IF
		IF DebugData.7 THEN Event[7].Text2 				:= CONCAT(Event[7].Text2, '|8');  END_IF
		Event[7].Text2 									:= CONCAT(Event[7].Text2, '|'); 
		
		Event[7](
			Flag	:= ShowEvent ,
			ConfirmTrig:= ConfirmTrig, 
			MsgId	:= 25, 
			pText3	:= ADR(DevTypeAndAddr))	;
	END_IF
	

//Events for EP1908 ****************************************************************)
IF Read.DebugDataMaxId > 16#10 THEN

	(* Fehler der Drehzahlueberwachung:Ueberdrehzahl *)
	Event[8].Flag 										:= Read.pDebugData^[16#13] <> 0;
	IF Event[8].Flag OR Event[8].Status.31
	THEN
		DebugData										:= Read.pDebugData^[16#13];
		Event[8].Text2									:= '';
		IF DebugData.0 THEN Event[8].Text2 				:= CONCAT(Event[8].Text2, '|1'); END_IF
		IF DebugData.1 THEN Event[8].Text2 				:= CONCAT(Event[8].Text2, '|2'); END_IF
		IF DebugData.2 THEN Event[8].Text2 				:= CONCAT(Event[8].Text2, '|3'); END_IF
		IF DebugData.3 THEN Event[8].Text2 				:= CONCAT(Event[8].Text2, '|4');  END_IF
		IF DebugData.4 THEN Event[8].Text2 				:= CONCAT(Event[8].Text2, '|5'); END_IF
		IF DebugData.5 THEN Event[8].Text2 				:= CONCAT(Event[8].Text2, '|6'); END_IF
		IF DebugData.6 THEN Event[8].Text2 				:= CONCAT(Event[8].Text2, '|7'); END_IF
		IF DebugData.7 THEN Event[8].Text2 				:= CONCAT(Event[8].Text2, '|8');  END_IF
		Event[8].Text2 									:= CONCAT(Event[8].Text2, '|'); 
		
		Event[8](
			Flag	:= ShowEvent ,
			ConfirmTrig:= ConfirmTrig, 
			MsgId	:= 26, 
			pText3	:= ADR(DevTypeAndAddr))	;
	END_IF
	
	(* Fehler in der Betriebsart: Two Channel Sync Velocity *)
	Event[9].Flag 										:= Read.pDebugData^[16#14] <> 0;
	IF Event[9].Flag OR Event[9].Status.31
	THEN
		DebugData										:= Read.pDebugData^[16#14];
		Event[9].Text2									:= '';
		IF DebugData.0 THEN Event[9].Text2 				:= CONCAT(Event[9].Text2, '|1+2'); END_IF
		IF DebugData.1 THEN Event[9].Text2 				:= CONCAT(Event[9].Text2, '|3+4'); END_IF
		IF DebugData.2 THEN Event[9].Text2 				:= CONCAT(Event[9].Text2, '|5+6'); END_IF
		IF DebugData.3 THEN Event[9].Text2 				:= CONCAT(Event[9].Text2, '|7+8');  END_IF
		Event[9].Text2 									:= CONCAT(Event[9].Text2, '|'); 
		
		Event[9](
			Flag	:= ShowEvent ,
			ConfirmTrig:= ConfirmTrig, 
			MsgId	:= 27, 
			pText3	:= ADR(DevTypeAndAddr))	;
	END_IF
	
	(* Fehler in der Betriebsart: Two Channel Sync Velocity UND Two Channel Encoder Velocity Control*)
	Event[10].Flag 										:= Read.pDebugData^[16#15] <> 0;
	IF Event[10].Flag OR Event[10].Status.31
	THEN
		DebugData										:= Read.pDebugData^[16#15];
		Event[10].Text2									:= '';
		IF DebugData.0 THEN Event[10].Text2 			:= CONCAT(Event[10].Text2, '|1+2'); END_IF
		IF DebugData.1 THEN Event[10].Text2 			:= CONCAT(Event[10].Text2, '|3+4'); END_IF
		IF DebugData.2 THEN Event[10].Text2 			:= CONCAT(Event[10].Text2, '|5+6'); END_IF
		IF DebugData.3 THEN Event[10].Text2 			:= CONCAT(Event[10].Text2, '|7+8');  END_IF
		Event[10].Text2 								:= CONCAT(Event[10].Text2, '|'); 
		
		Event[10](
			Flag	:= ShowEvent ,
			ConfirmTrig:= ConfirmTrig, 
			MsgId	:= 28, 
			pText3	:= ADR(DevTypeAndAddr))	;
	END_IF
END_IF

(************************************************************************************)
END_METHOD

END_FUNCTION_BLOCK

// POUs/Safety/Diag/SafetyIODeviceDiagRead
{attribute 'no_check'}
{attribute 'enable_dynamic_creation'}
FUNCTION_BLOCK SafetyIODeviceDiagRead EXTENDS FbBase
VAR CONSTANT
	bitTwinSAFETerm											:	BYTE := 0; //Ex1918,ELx9xx, etc. (2nd generation of TwinSAFE devices with CoE Index 10F3 Diag History included)
	bitSafetyTerm											:	BYTE := 1; //EL1904,EL2904,EK1914,EP1908 (Diagnoses provided via CoE Index 0x800E FSOE Internal Data, Debug 1..x) 
 	bitAX58xx												:	BYTE := 2; //AX5805,AX5806 (Diag via CoE index 0xFA10)
END_VAR
VAR_INPUT
	EcMasterDevId											:	UINT;	//EtherCAT Master DevId
END_VAR                 									
VAR_OUTPUT              									 
	AdsAddr											AT %I*	:	AMSADDR; //Link to terminal/box/device AMS Net Addr.
	{attribute 'displaymode':='binary'}
	MsgInfoDiag										AT %I*	:	USINT; 	//Link to connection messagediag of EL69xx (Needs to be enabled for alias of device)
//	{attribute 'displaymode':='hexadecimal'}
//	MsgInfoState									AT %I*	:	USINT; 	//Link to connection message state of EL69xx (Needs to be enabled for alias of device)	
	DevType													:	STRING(15); //CoE index 1008 / e.g. EL1908, EP1957-0022, etc...
	Name													:	STRING(31);	//Device name as defined in system manager configuration								
	FSOEAddr												:	WORD; //CoE index 0xF980
	DiagMsgSeverity											:	UINT; //Info (0) Warning (1) or Error (2)
	{attribute 'displaymode':='hexadecimal'}
	DiagMsgTextId											: 	UINT; //CoE Index 10F3 newest diagnoses message TextID (xyzz -> X =Type | y = Source | zz = Message ID)
	{attribute 'displaymode':='hexadecimal'}
	pDebugData												:	POINTER TO ARRAY[0..64] OF WORD; //Pointer to CoE index 0x800E - FSOE Internal Data - Debug 1-x for diag of "Safety Terminals" (or CoE Index 0xFA10 for AX58xx)
	DebugDataMaxId											:	UINT; //Max index for pointer pDebugData to array of word (Debug 1..x) if 0 data are invalid		
END_VAR                 									

VAR(* internal *)    
	{attribute 'displaymode':='bin'}
	DevCategory												:	BYTE;
	IOF_GetBoxNameByAddr									:	IOF_GetBoxNameByAddr := (TMOUT	:= DEFAULT_ADS_TIMEOUT);
	EcCoEReadDiagMsg										:	EcCoEReadNewestDiagMsg ;              									
	EcCoESdoReadEx											:	FB_EcCoESdoReadEx := (tTimeout := DEFAULT_ADS_TIMEOUT);       
	i														:	INT;  								                            	
END_VAR
(*
Tabelle 2-4: Diagnose-Informationen einer Connection
Wert Beschreibung
xxxx 0001 invalid command
xxxx 0010 unknown command
xxxx 0011 invalid connection ID
xxxx 0100 invalid CRC
xxxx 0101 Watchdog run out of time
xxxx 0110 invalid FSoE-Adress
xxxx 0111 invalid data
xxxx 1000 invalid length of communicatoin parameter Kommunikationsparameterlänge
xxxx 1001 invalid communicatoin parameter
xxxx 1010 invalid operator parameter length
xxxx 1011 invalid operator parameter
xxxx 1100 FSoE Master Reset
xxxx 1101 Module fault on slave detected with activated option "Modulfault is ComError"
xxxx 1110 Module fault on EL290x at activated with option "Error achnowledge active"
xxxx 1111 Slave not started or unexpected error argument

xxx1 xxxx FSoE Slave error detected
xx1x xxxx FSoE Slave notifies Failsafe Value active
x1xx xxxx StartUp
1xxx xxxx FSoE Master notifies Failsafe Value active
*)

(* IO Safety Terminal Status Diag		V2.0	*)
(************************************************)

(* Trigger to read diag **********************************************)
	rtExecute(CLK := Execute);
	
(* Read adress and type ***********************************************)
	CASE state OF
	0:
		Busy 												:= FALSE;
		IF NOT Execute
		THEN
			Done											:= FALSE;
			Error											:= FALSE;
			ErrorId											:= 0;					
		END_IF
		
		IF rtExecute.Q
		THEN
			Busy 											:= TRUE;
			Done											:= FALSE;
			Error											:= FALSE;
			ErrorId											:= 0;
			DiagMsgTextId									:= 0;
			DiagMsgSeverity									:= 0;

			EcCoESdoReadEx(bExecute := FALSE, bCompleteAccess := FALSE);
			IOF_GetBoxNameByAddr(Start := FALSE);
			EcCoEReadDiagMsg(Execute := FALSE);
			
			IF DevCategory.bitTwinSAFETerm
			THEN
				state 										:= 10;	
			ELSIF DevCategory.bitSafetyTerm
			THEN
				state 										:= SEL(DebugDataMaxId = 0, 21, 20);
			ELSIF DevCategory.bitAX58xx				
			THEN 
				state 										:= 30;
				
			ELSE //Read more device information 
				state										:= state + 1;				
			END_IF
		
		END_IF

	1: (* read FSOE adress *)
		EcCoESdoReadEx(
			sNetId			:= F_CreateAmsNetId(nIds := AdsAddr.netId ),
			nSlaveAddr		:= AdsAddr.port,
			nSubIndex		:= 16#1,
			nIndex			:= 16#F980,
			pDstBuf			:= ADR(FSOEAddr),
			cbBufLen		:= SIZEOF(FSOEAddr),
			bExecute		:= TRUE,
			tTimeout		:=  (* Default *),
			bCompleteAccess	:= ,
			bBusy			=> ,
			bError			=> ,
			nErrId			=> );
			
		IF NOT EcCoESdoReadEx.bBusy
		THEN
			IF EcCoESdoReadEx.bError 
			THEN
				Busy 										:= FALSE;
				Error										:= TRUE;
				ErrorId										:= EcCoESdoReadEx.nErrId;
				DiagMsgTextId								:= TO_UINT(state);
				state										:= 0;
			ELSE      									
				state 										:= state + 1;
			END_IF
			EcCoESdoReadEx(bExecute := FALSE);
		END_IF

	2: //Ready name from system manager configuration
		IOF_GetBoxNameByAddr(
			NETID		:='' , (* Local *)
			DEVICEID	:= UINT_TO_UDINT(EcMasterDevId) ,
			BOXADDR		:= AdsAddr.port ,
			START		:= EcMasterDevId <> 0,
			BOXNAME		=> );
			
		IF NOT IOF_GetBoxNameByAddr.Busy
		THEN
			IF IOF_GetBoxNameByAddr.Err 
			THEN
				Busy 										:= FALSE;
				Error										:= TRUE;
				ErrorId										:= IOF_GetBoxNameByAddr.ERRID;
				DiagMsgTextId								:= TO_UINT(state);
				state										:= 0;
			ELSIF IOF_GetBoxNameByAddr.Start
			THEN
				state 										:= state + 1;
			ELSE //No box name to read
				Name										:= CONCAT('EtherCAT Addr.',TO_STRING(AdsAddr.port));
			END_IF
			IOF_GetBoxNameByAddr(START := FALSE);
		END_IF
		
	3:  (* read device name e.g. EL1904 *)
		EcCoESdoReadEx(bExecute	:= TRUE, nIndex	:= 16#1008, nSubIndex := 16#0, pDstBuf := ADR(DevType),cbBufLen	:= SIZEOF(DevType));

		IF NOT EcCoESdoReadEx.bBusy
		THEN
			IF EcCoESdoReadEx.bError 
			THEN
				Busy 										:= FALSE;
				Error										:= TRUE;
				ErrorId										:= EcCoESdoReadEx.nErrId;
				DiagMsgTextId								:= TO_UINT(state);
				state										:= 0;
			ELSE       
				 //Delte type from name if in brakets 
				Name										:= DELETE(IOF_GetBoxNameByAddr.BOXNAME, LEN(DevType) + 2 , FIND(IOF_GetBoxNameByAddr.BOXNAME,DevType) - 1);
                             	
				IF DevType = 'AX5806' OR_ELSE DevType = 'AX5805'
				THEN
					DevCategory.bitAX58xx					:= TRUE;
					state 									:= 30;
				ELSIF DevType = 'EL1904' OR_ELSE DevType = 'EL2904' OR_ELSE DevType = 'EK1914' OR_ELSE DevType = 'EP1908'
				THEN
					DevCategory.bitSafetyTerm 				:= TRUE;
					state 									:= SEL(DebugDataMaxId = 0, 21, 20);
				ELSE
					DevCategory.bitTwinSAFETerm				:= TRUE;
					state 									:= 10;
				END_IF
				
			END_IF
			EcCoESdoReadEx(bExecute := FALSE);
		END_IF

	(* Read diagnoses latest entry from diag history ***********************************)	
	10: 
		EcCoEReadDiagMsg(Execute := TRUE, AdsAddr := AdsAddr);
		IF NOT EcCoEReadDiagMsg.Busy
		THEN
			IF EcCoEReadDiagMsg.Error 
			THEN
				Busy 										:= FALSE;
				Error										:= TRUE;
				ErrorId										:= EcCoEReadDiagMsg.ErrorID;
				DiagMsgTextId								:= TO_UINT(state);
				state										:= 0;				
			ELSE
				DiagMsgTextId								:= EcCoEReadDiagMsg.MsgId;
				DiagMsgSeverity								:= EcCoEReadDiagMsg.MsgSeverity;
				Done										:= TRUE;
				Busy										:= FALSE;
				State										:= 0;
			END_IF
		END_IF
		
	(* Read lenght of 0x800E:0 FSOE internal data.Debug terminal *********************************)
	20:
		EcCoESdoReadEx(bExecute	:= DebugDataMaxId = 0, nIndex	:= 16#800E, nSubIndex := 16#0, pDstBuf := ADR(DebugDataMaxId),cbBufLen	:= SIZEOF(DebugDataMaxId));

